KUKA KRL program: EPS_2_25716_MHCR05_A_20250828081216.src

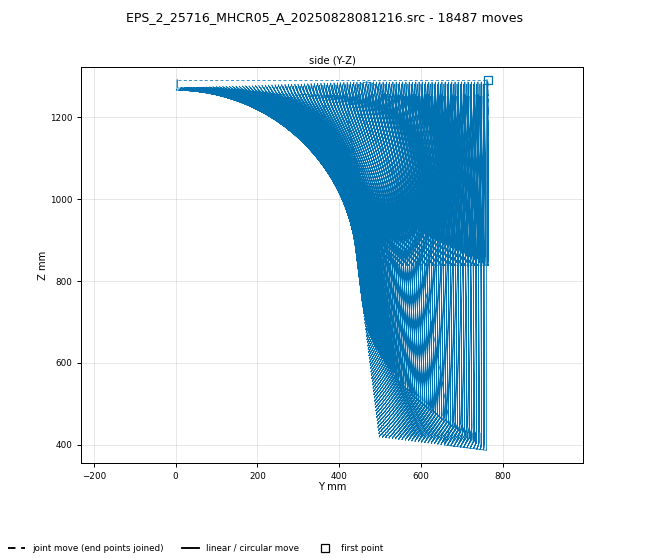
[picture p0: tool path of EPS_2_25716_MHCR05_A_20250828081216.src, 18487 of 18489 moves have a stored position in this frame; points joined in program order, loops and branches not executed]
&ACCESS RVP
&REL 4
&COMMENT QRS 19112012
&PARAM EDITMASK = *
DEF PART()
EXT BAS (BAS_COMMAND :IN,REAL :IN )
INT I
BAS (#INITMOV,0 )

;KUKA QRS Post kuka4.cps  Date:22-06-2017 !

File_ID=2804

QRS_PRE_INIT()

;Init var - Until changes are made in qrs_pre_init
Outlet_Square_prg=0
Inlet_1_Square_prg=0
Inlet_2_Square_prg=0
Inlet_3_Square_prg=0
Inlet_4_Square_prg=0
Inlet_5_Square_prg=0

Outlet_1={X 0.000, Y 457.000, Z 863.000, B 0.000, E1 0.000 }
Inlet_1={X 0.000, Y 457.000, Z 833.000, B 0.000, E1 180.000 }
Outlet_1_type=838
Inlet_1_type=838
;QRS#1=Sidecore dimensions
;QRS#2=825-33" Concrete
;QRS#3=825-33" Concrete
;QRS#4=
;QRS#5=
;QRS#6=
;QRS#7=
;QRS#8=
;QRS#9=S306-46
;QRS#10=S306-46
;QRS#11=
;QRS#12=
;QRS#13=
;QRS#14=
;QRS#15=
;QRS#16=1524x152x1753 5,75'
;QRS#17=EPS Height
;QRS#18=1282
;QRS#19=*
;QRS#20= UPDATED VERSION 22-06-2017
;QRS#21=*
Outlet_Square=0650
Inlet_1_Square=0650
Inlet_2_Square=0
Inlet_3_Square=0
Inlet_4_Square=0
Inlet_5_Square=0
Mill_Square=1
Outlet_Square_Prg=267
Inlet_1_Square_prg=267

QRS_INIT()

$ADVANCE=5

; T1
PTP {E1 177.513,E2 177.513}
PTP {X 0,Y 762.785,A -85,B 0,C 180,E1 177.513,E2 177.513,E3 0,E4 0,E5 0,E6 0}
QRS_SPEED_INIT()
LIN {X 0,Y 762.785,Z 1292,A -85,B 0,C 180,E1 177.513,E2 177.513,E3 0,E4 0,E5 0,E6 0} C_VEL
LIN {X 0,Y 762.785,Z 841.06,A -85,B 0,C 180,E1 177.513,E2 177.513} C_VEL
LIN {X 0,Y 762.866,Z 839.06,A -85,B 0,C 180,E1 177.663,E2 177.663} C_VEL
LIN {X 0,Y 763.878,Z 839.06,A -85,B 0,C 180,E1 179.063,E2 179.063} C_VEL
LIN {X 0,Y 763.781,Z 839.06,A -85,B 0,C 180,E1 186.577,E2 186.577} C_VEL
LIN {X 0,Y 763.753,Z 839.06,A -85,B 0,C 180,E1 194.208,E2 194.208} C_VEL
LIN {X 0,Y 763.775,Z 839.06,A -85,B 0,C 180,E1 202.107,E2 202.107} C_VEL
LIN {X 0,Y 762.947,Z 839.06,A -85,B 0,C 180,E1 208.361,E2 208.361} C_VEL
LIN {X 0,Y 763.678,Z 839.06,A -85,B 0,C 180,E1 209.865,E2 209.865} C_VEL
LIN {X 0,Y 763.751,Z 839.06,A -85,B 0,C 180,E1 217.259,E2 217.259} C_VEL
LIN {X 0,Y 762.19,Z 839.06,A -85,B 0,C 180,E1 222.241,E2 222.241} C_VEL
LIN {X 0,Y 763.489,Z 839.06,A -85,B 0,C 180,E1 224.736,E2 224.736} C_VEL
LIN {X 0,Y 763.718,Z 839.06,A -85,B 0,C 180,E1 225.289,E2 225.289} C_VEL
LIN {X 0,Y 763.691,Z 839.06,A -85,B 0,C 180,E1 233.306,E2 233.306} C_VEL
LIN {X 0,Y 763.599,Z 839.06,A -85,B 0,C 180,E1 233.585,E2 233.585} C_VEL
LIN {X 0,Y 763.105,Z 842.178,A -85,B 0,C 180,E1 233.692,E2 233.692} C_VEL
LIN {X 0,Y 763.151,Z 902.432,A -85,B 0,C 180,E1 234.391,E2 234.391} C_VEL
LIN {X 0,Y 763.569,Z 919.488,A -85,B 0,C 180,E1 234.674,E2 234.674} C_VEL
LIN {X 0,Y 763.689,Z 936.684,A -85,B 0,C 180,E1 235.004,E2 235.004} C_VEL
LIN {X 0,Y 763.627,Z 953.994,A -85,B 0,C 180,E1 235.388,E2 235.388} C_VEL
LIN {X 0,Y 763.298,Z 971.622,A -85,B 0,C 180,E1 235.836,E2 235.836} C_VEL
LIN {X 0,Y 763.66,Z 994.06,A -85,B 0,C 180,E1 236.546,E2 236.546} C_VEL
LIN {X 0,Y 763.665,Z 1012.884,A -85,B 0,C 180,E1 237.214,E2 237.214} C_VEL
LIN {X 0,Y 763.649,Z 1032.465,A -85,B 0,C 180,E1 238,E2 238} C_VEL
LIN {X 0,Y 763.47,Z 1045.091,A -85,B 0,C 180,E1 238.553,E2 238.553} C_VEL
LIN {X 0,Y 763.557,Z 1053.715,A -85,B 0,C 180,E1 238.962,E2 238.962} C_VEL
LIN {X 0,Y 763.507,Z 1068.148,A -85,B 0,C 180,E1 239.675,E2 239.675} C_VEL
LIN {X 0,Y 763.465,Z 1085.374,A -85,B 0,C 180,E1 240.61,E2 240.61} C_VEL
LIN {X 0,Y 763.616,Z 1101.645,A -85,B 0,C 180,E1 241.581,E2 241.581} C_VEL
LIN {X 0,Y 763.575,Z 1117.447,A -85,B 0,C 180,E1 242.599,E2 242.599} C_VEL
LIN {X 0,Y 763.286,Z 1132.483,A -85,B 0,C 180,E1 243.639,E2 243.639} C_VEL
LIN {X 0,Y 763.185,Z 1147.05,A -85,B 0,C 180,E1 244.739,E2 244.739} C_VEL
LIN {X 0,Y 763.452,Z 1160.517,A -85,B 0,C 180,E1 245.849,E2 245.849} C_VEL
LIN {X 0,Y 763.696,Z 1173.568,A -85,B 0,C 180,E1 247.008,E2 247.008} C_VEL
LIN {X 0,Y 763.172,Z 1187.049,A -85,B 0,C 180,E1 248.284,E2 248.284} C_VEL
LIN {X 0,Y 762.923,Z 1198.82,A -85,B 0,C 180,E1 249.499,E2 249.499} C_VEL
LIN {X 0,Y 763.252,Z 1210.585,A -85,B 0,C 180,E1 250.839,E2 250.839} C_VEL
LIN {X 0,Y 763.819,Z 1221.039,A -85,B 0,C 180,E1 252.14,E2 252.14} C_VEL
LIN {X 0,Y 763.048,Z 1231.864,A -85,B 0,C 180,E1 253.594,E2 253.594} C_VEL
LIN {X 0,Y 762.736,Z 1241.602,A -85,B 0,C 180,E1 255.059,E2 255.059} C_VEL
LIN {X 0,Y 763.109,Z 1249.379,A -85,B 0,C 180,E1 256.364,E2 256.364} C_VEL
LIN {X 0,Y 763.845,Z 1256.57,A -85,B 0,C 180,E1 257.724,E2 257.724} C_VEL
LIN {X 0,Y 762.883,Z 1264.428,A -85,B 0,C 180,E1 259.384,E2 259.384} C_VEL
LIN {X 0,Y 762.623,Z 1269.209,A -85,B 0,C 180,E1 260.572,E2 260.572} C_VEL
LIN {X 0,Y 762.835,Z 1272.583,A -85,B 0,C 180,E1 261.525,E2 261.525} C_VEL
LIN {X 0,Y 763.28,Z 1275.723,A -85,B 0,C 180,E1 262.478,E2 262.478} C_VEL
LIN {X 0,Y 763.858,Z 1278.353,A -85,B 0,C 180,E1 263.428,E2 263.428} C_VEL
LIN {X 0,Y 763.258,Z 1280.666,A -85,B 0,C 180,E1 264.366,E2 264.366} C_VEL
LIN {X 0,Y 762.774,Z 1282.62,A -85,B 0,C 180,E1 265.305,E2 265.305} C_VEL
LIN {X 0,Y 762.587,Z 1284.207,A -85,B 0,C 180,E1 266.245,E2 266.245} C_VEL
LIN {X 0,Y 762.778,Z 1285.378,A -85,B 0,C 180,E1 267.186,E2 267.186} C_VEL
LIN {X 0,Y 763.829,Z 1286.67,A -85,B 0,C 180,E1 269.066,E2 269.066} C_VEL
LIN {X 0,Y 762.793,Z 1286.715,A -85,B 0,C 180,E1 270.942,E2 270.942} C_VEL
LIN {X 0,Y 762.612,Z 1286.489,A -85,B 0,C 180,E1 271.58,E2 271.58} C_VEL
LIN {X 0,Y 762.793,Z 1285.372,A -85,B 0,C 180,E1 272.82,E2 272.82} C_VEL
LIN {X 0,Y 763.264,Z 1284.181,A -85,B 0,C 180,E1 273.758,E2 273.758} C_VEL
LIN {X 0,Y 763.868,Z 1282.57,A -85,B 0,C 180,E1 274.695,E2 274.695} C_VEL
LIN {X 0,Y 763.015,Z 1279.579,A -85,B 0,C 180,E1 276.114,E2 276.114} C_VEL
LIN {X 0,Y 762.631,Z 1275.706,A -85,B 0,C 180,E1 277.536,E2 277.536} C_VEL
LIN {X 0,Y 763.011,Z 1270.959,A -85,B 0,C 180,E1 278.954,E2 278.954} C_VEL
LIN {X 0,Y 763.87,Z 1265.354,A -85,B 0,C 180,E1 280.37,E2 280.37} C_VEL
LIN {X 0,Y 763.474,Z 1262.202,A -85,B 0,C 180,E1 281.092,E2 281.092} C_VEL
LIN {X 0,Y 762.849,Z 1256.532,A -85,B 0,C 180,E1 282.299,E2 282.299} C_VEL
LIN {X 0,Y 762.722,Z 1249.063,A -85,B 0,C 180,E1 283.698,E2 283.698} C_VEL
LIN {X 0,Y 763.275,Z 1240.923,A -85,B 0,C 180,E1 285.043,E2 285.043} C_VEL
LIN {X 0,Y 763.758,Z 1235.327,A -85,B 0,C 180,E1 285.873,E2 285.873} C_VEL
LIN {X 0,Y 763.633,Z 1231.816,A -85,B 0,C 180,E1 286.4,E2 286.4} C_VEL
LIN {X 0,Y 762.911,Z 1220.984,A -85,B 0,C 180,E1 287.889,E2 287.889} C_VEL
LIN {X 0,Y 762.868,Z 1209,A -85,B 0,C 180,E1 289.358,E2 289.358} C_VEL
LIN {X 0,Y 763.421,Z 1197.407,A -85,B 0,C 180,E1 290.64,E2 290.64} C_VEL
LIN {X 0,Y 763.771,Z 1189.172,A -85,B 0,C 180,E1 291.478,E2 291.478} C_VEL
LIN {X 0,Y 763.561,Z 1182.825,A -85,B 0,C 180,E1 292.116,E2 292.116} C_VEL
LIN {X 0,Y 763.219,Z 1172.077,A -85,B 0,C 180,E1 293.142,E2 293.142} C_VEL
LIN {X 0,Y 763.156,Z 1158.949,A -85,B 0,C 180,E1 294.293,E2 294.293} C_VEL
LIN {X 0,Y 763.463,Z 1145.228,A -85,B 0,C 180,E1 295.394,E2 295.394} C_VEL
LIN {X 0,Y 763.662,Z 1130.565,A -85,B 0,C 180,E1 296.486,E2 296.486} C_VEL
LIN {X 0,Y 763.467,Z 1114.323,A -85,B 0,C 180,E1 297.612,E2 297.612} C_VEL
LIN {X 0,Y 763.401,Z 1098.789,A -85,B 0,C 180,E1 298.602,E2 298.602} C_VEL
LIN {X 0,Y 763.564,Z 1082.344,A -85,B 0,C 180,E1 299.557,E2 299.557} C_VEL
LIN {X 0,Y 763.601,Z 1066.411,A -85,B 0,C 180,E1 300.413,E2 300.413} C_VEL
LIN {X 0,Y 763.622,Z 1047.439,A -85,B 0,C 180,E1 301.337,E2 301.337} C_VEL
LIN {X 0,Y 763.594,Z 1028.686,A -85,B 0,C 180,E1 302.161,E2 302.161} C_VEL
LIN {X 0,Y 763.579,Z 1010.173,A -85,B 0,C 180,E1 302.89,E2 302.89} C_VEL
LIN {X 0,Y 763.358,Z 997.463,A -85,B 0,C 180,E1 303.349,E2 303.349} C_VEL
LIN {X 0,Y 763.576,Z 988.896,A -85,B 0,C 180,E1 303.623,E2 303.623} C_VEL
LIN {X 0,Y 763.726,Z 970.079,A -85,B 0,C 180,E1 304.185,E2 304.185} C_VEL
LIN {X 0,Y 763.711,Z 953.48,A -85,B 0,C 180,E1 304.621,E2 304.621} C_VEL
LIN {X 0,Y 763.519,Z 936.23,A -85,B 0,C 180,E1 305.015,E2 305.015} C_VEL
LIN {X 0,Y 763.194,Z 924.975,A -85,B 0,C 180,E1 305.251,E2 305.251} C_VEL
LIN {X 0,Y 763.49,Z 908.084,A -85,B 0,C 180,E1 305.51,E2 305.51} C_VEL
LIN {X 0,Y 763.502,Z 896.075,A -85,B 0,C 180,E1 305.669,E2 305.669} C_VEL
LIN {X 0,Y 763.101,Z 839.511,A -85,B 0,C 180,E1 306.339,E2 306.339} C_VEL
LIN {X 0,Y 763.718,Z 839.06,A -85,B 0,C 180,E1 306.442,E2 306.442} C_VEL
LIN {X 0,Y 763.692,Z 839.06,A -85,B 0,C 180,E1 306.694,E2 306.694} C_VEL
LIN {X 0,Y 763.713,Z 839.06,A -85,B 0,C 180,E1 314.721,E2 314.721} C_VEL
LIN {X 0,Y 763.497,Z 839.06,A -85,B 0,C 180,E1 315.265,E2 315.265} C_VEL
LIN {X 0,Y 762.413,Z 839.06,A -85,B 0,C 180,E1 320.391,E2 320.391} C_VEL
LIN {X 0,Y 763.779,Z 839.06,A -85,B 0,C 180,E1 322.742,E2 322.742} C_VEL
LIN {X 0,Y 763.789,Z 839.06,A -85,B 0,C 180,E1 329.521,E2 329.521} C_VEL
LIN {X 0,Y 763.786,Z 839.06,A -85,B 0,C 180,E1 335.855,E2 335.855} C_VEL
LIN {X 0,Y 763.81,Z 839.06,A -85,B 0,C 180,E1 343.85,E2 343.85} C_VEL
LIN {X 0,Y 763.85,Z 839.06,A -85,B 0,C 180,E1 351.533,E2 351.533} C_VEL
LIN {X 0,Y 763.887,Z 839.06,A -85,B 0,C 180,E1 359.063,E2 359.063} C_VEL
LIN {X 0,Y 763.839,Z 839.06,A -85,B 0,C 180,E1 366.576,E2 366.576} C_VEL
LIN {X 0,Y 763.861,Z 839.06,A -85,B 0,C 180,E1 374.206,E2 374.206} C_VEL
LIN {X 0,Y 763.821,Z 839.06,A -85,B 0,C 180,E1 382.105,E2 382.105} C_VEL
LIN {X 0,Y 762.949,Z 839.06,A -85,B 0,C 180,E1 388.361,E2 388.361} C_VEL
LIN {X 0,Y 763.665,Z 839.06,A -85,B 0,C 180,E1 389.85,E2 389.85} C_VEL
LIN {X 0,Y 763.783,Z 839.06,A -85,B 0,C 180,E1 397.257,E2 397.257} C_VEL
LIN {X 0,Y 762.287,Z 839.06,A -85,B 0,C 180,E1 402.459,E2 402.459} C_VEL
LIN {X 0,Y 763.519,Z 839.06,A -85,B 0,C 180,E1 404.734,E2 404.734} C_VEL
LIN {X 0,Y 763.736,Z 839.06,A -85,B 0,C 180,E1 405.281,E2 405.281} C_VEL
LIN {X 0,Y 763.707,Z 839.06,A -85,B 0,C 180,E1 413.304,E2 413.304} C_VEL
LIN {X 0,Y 763.661,Z 839.06,A -85,B 0,C 180,E1 413.601,E2 413.601} C_VEL
LIN {X 0,Y 761.689,Z 839.06,A -85,B 0,C 180,E1 413.812,E2 413.812} C_VEL
LIN {X 0,Y 761.812,Z 840.818,A -85,B 0,C 180,E1 413.903,E2 413.903} C_VEL
LIN {X 0,Y 762.77,Z 843.615,A -85,B 0,C 180,E1 413.987,E2 413.987} C_VEL
LIN {X 0,Y 763.13,Z 845.592,A -85,B 0,C 180,E1 414.029,E2 414.029} C_VEL
LIN {X 0,Y 763.65,Z 875.73,A -85,B 0,C 180,E1 414.419,E2 414.419} C_VEL
LIN {X 0,Y 763.658,Z 892.175,A -85,B 0,C 180,E1 414.679,E2 414.679} C_VEL
LIN {X 0,Y 763.408,Z 909.107,A -85,B 0,C 180,E1 414.995,E2 414.995} C_VEL
LIN {X 0,Y 763.241,Z 916.55,A -85,B 0,C 180,E1 415.149,E2 415.149} C_VEL
LIN {X 0,Y 763.606,Z 932.664,A -85,B 0,C 180,E1 415.562,E2 415.562} C_VEL
LIN {X 0,Y 763.666,Z 945.84,A -85,B 0,C 180,E1 415.934,E2 415.934} C_VEL
LIN {X 0,Y 763.644,Z 964.876,A -85,B 0,C 180,E1 416.529,E2 416.529} C_VEL
LIN {X 0,Y 763.371,Z 982.796,A -85,B 0,C 180,E1 417.152,E2 417.152} C_VEL
LIN {X 0,Y 763.602,Z 1002.249,A -85,B 0,C 180,E1 417.944,E2 417.944} C_VEL
LIN {X 0,Y 763.603,Z 1020.397,A -85,B 0,C 180,E1 418.756,E2 418.756} C_VEL
LIN {X 0,Y 763.645,Z 1038.535,A -85,B 0,C 180,E1 419.657,E2 419.657} C_VEL
LIN {X 0,Y 763.579,Z 1054.594,A -85,B 0,C 180,E1 420.524,E2 420.524} C_VEL
LIN {X 0,Y 763.423,Z 1071.141,A -85,B 0,C 180,E1 421.496,E2 421.496} C_VEL
LIN {X 0,Y 763.34,Z 1087.981,A -85,B 0,C 180,E1 422.582,E2 422.582} C_VEL
LIN {X 0,Y 763.549,Z 1102.977,A -85,B 0,C 180,E1 423.641,E2 423.641} C_VEL
LIN {X 0,Y 763.649,Z 1117.051,A -85,B 0,C 180,E1 424.71,E2 424.71} C_VEL
LIN {X 0,Y 763.257,Z 1130.941,A -85,B 0,C 180,E1 425.835,E2 425.835} C_VEL
LIN {X 0,Y 763.008,Z 1143.961,A -85,B 0,C 180,E1 426.978,E2 426.978} C_VEL
LIN {X 0,Y 763.296,Z 1157.072,A -85,B 0,C 180,E1 428.245,E2 428.245} C_VEL
LIN {X 0,Y 763.8,Z 1169.152,A -85,B 0,C 180,E1 429.516,E2 429.516} C_VEL
LIN {X 0,Y 763.197,Z 1180.742,A -85,B 0,C 180,E1 430.812,E2 430.812} C_VEL
LIN {X 0,Y 762.792,Z 1191.318,A -85,B 0,C 180,E1 432.108,E2 432.108} C_VEL
LIN {X 0,Y 763.104,Z 1202.116,A -85,B 0,C 180,E1 433.588,E2 433.588} C_VEL
LIN {X 0,Y 763.757,Z 1210.687,A -85,B 0,C 180,E1 434.883,E2 434.883} C_VEL
LIN {X 0,Y 763.675,Z 1213.295,A -85,B 0,C 180,E1 435.315,E2 435.315} C_VEL
LIN {X 0,Y 763.015,Z 1219.935,A -85,B 0,C 180,E1 436.42,E2 436.42} C_VEL
LIN {X 0,Y 762.583,Z 1227.944,A -85,B 0,C 180,E1 437.937,E2 437.937} C_VEL
LIN {X 0,Y 762.996,Z 1234.58,A -85,B 0,C 180,E1 439.379,E2 439.379} C_VEL
LIN {X 0,Y 763.697,Z 1239.36,A -85,B 0,C 180,E1 440.579,E2 440.579} C_VEL
LIN {X 0,Y 763.674,Z 1241.105,A -85,B 0,C 180,E1 441.053,E2 441.053} C_VEL
LIN {X 0,Y 762.88,Z 1245.837,A -85,B 0,C 180,E1 442.467,E2 442.467} C_VEL
LIN {X 0,Y 762.627,Z 1249.69,A -85,B 0,C 180,E1 443.882,E2 443.882} C_VEL
LIN {X 0,Y 763.151,Z 1252.687,A -85,B 0,C 180,E1 445.3,E2 445.3} C_VEL
LIN {X 0,Y 763.839,Z 1254.408,A -85,B 0,C 180,E1 446.388,E2 446.388} C_VEL
LIN {X 0,Y 763.401,Z 1255.391,A -85,B 0,C 180,E1 447.182,E2 447.182} C_VEL
LIN {X 0,Y 762.542,Z 1256.734,A -85,B 0,C 180,E1 449.058,E2 449.058} C_VEL
LIN {X 0,Y 762.958,Z 1256.698,A -85,B 0,C 180,E1 450.935,E2 450.935} C_VEL
LIN {X 0,Y 763.557,Z 1255.31,A -85,B 0,C 180,E1 452.811,E2 452.811} C_VEL
LIN {X 0,Y 762.975,Z 1254.137,A -85,B 0,C 180,E1 453.753,E2 453.753} C_VEL
LIN {X 0,Y 762.645,Z 1252.533,A -85,B 0,C 180,E1 454.696,E2 454.696} C_VEL
LIN {X 0,Y 762.762,Z 1249.484,A -85,B 0,C 180,E1 456.11,E2 456.11} C_VEL
LIN {X 0,Y 763.538,Z 1245.587,A -85,B 0,C 180,E1 457.52,E2 457.52} C_VEL
LIN {X 0,Y 763.844,Z 1244.019,A -85,B 0,C 180,E1 457.99,E2 457.99} C_VEL
LIN {X 0,Y 763.275,Z 1240.83,A -85,B 0,C 180,E1 458.944,E2 458.944} C_VEL
LIN {X 0,Y 762.602,Z 1234.243,A -85,B 0,C 180,E1 460.62,E2 460.62} C_VEL
LIN {X 0,Y 762.993,Z 1226.33,A -85,B 0,C 180,E1 462.29,E2 462.29} C_VEL
LIN {X 0,Y 763.73,Z 1219.455,A -85,B 0,C 180,E1 463.566,E2 463.566} C_VEL
LIN {X 0,Y 763.759,Z 1217.556,A -85,B 0,C 180,E1 463.884,E2 463.884} C_VEL
LIN {X 0,Y 763.136,Z 1210.866,A -85,B 0,C 180,E1 465.01,E2 465.01} C_VEL
LIN {X 0,Y 762.705,Z 1201.563,A -85,B 0,C 180,E1 466.414,E2 466.414} C_VEL
LIN {X 0,Y 763.094,Z 1189.694,A -85,B 0,C 180,E1 468.001,E2 468.001} C_VEL
LIN {X 0,Y 763.767,Z 1179.038,A -85,B 0,C 180,E1 469.285,E2 469.285} C_VEL
LIN {X 0,Y 763.28,Z 1167.08,A -85,B 0,C 180,E1 470.632,E2 470.632} C_VEL
LIN {X 0,Y 762.97,Z 1155.209,A -85,B 0,C 180,E1 471.862,E2 471.862} C_VEL
LIN {X 0,Y 763.232,Z 1141.649,A -85,B 0,C 180,E1 473.135,E2 473.135} C_VEL
LIN {X 0,Y 763.679,Z 1128.165,A -85,B 0,C 180,E1 474.294,E2 474.294} C_VEL
LIN {X 0,Y 763.562,Z 1116.121,A -85,B 0,C 180,E1 475.278,E2 475.278} C_VEL
LIN {X 0,Y 763.276,Z 1100.026,A -85,B 0,C 180,E1 476.492,E2 476.492} C_VEL
LIN {X 0,Y 763.361,Z 1084.775,A -85,B 0,C 180,E1 477.542,E2 477.542} C_VEL
LIN {X 0,Y 763.577,Z 1068.971,A -85,B 0,C 180,E1 478.539,E2 478.539} C_VEL
LIN {X 0,Y 763.632,Z 1051.912,A -85,B 0,C 180,E1 479.532,E2 479.532} C_VEL
LIN {X 0,Y 763.542,Z 1035.674,A -85,B 0,C 180,E1 480.407,E2 480.407} C_VEL
LIN {X 0,Y 763.571,Z 1017.254,A -85,B 0,C 180,E1 481.302,E2 481.302} C_VEL
LIN {X 0,Y 763.523,Z 998.236,A -85,B 0,C 180,E1 482.137,E2 482.137} C_VEL
LIN {X 0,Y 763.43,Z 991.336,A -85,B 0,C 180,E1 482.416,E2 482.416} C_VEL
LIN {X 0,Y 763.663,Z 979.229,A -85,B 0,C 180,E1 482.874,E2 482.874} C_VEL
LIN {X 0,Y 763.696,Z 961.114,A -85,B 0,C 180,E1 483.504,E2 483.504} C_VEL
LIN {X 0,Y 763.649,Z 940.7,A -85,B 0,C 180,E1 484.127,E2 484.127} C_VEL
LIN {X 0,Y 763.287,Z 923.063,A -85,B 0,C 180,E1 484.608,E2 484.608} C_VEL
LIN {X 0,Y 763.424,Z 916.043,A -85,B 0,C 180,E1 484.763,E2 484.763} C_VEL
LIN {X 0,Y 763.72,Z 898.672,A -85,B 0,C 180,E1 485.108,E2 485.108} C_VEL
LIN {X 0,Y 763.762,Z 883.162,A -85,B 0,C 180,E1 485.376,E2 485.376} C_VEL
LIN {X 0,Y 763.655,Z 867.28,A -85,B 0,C 180,E1 485.601,E2 485.601} C_VEL
LIN {X 0,Y 763.073,Z 839.454,A -85,B 0,C 180,E1 485.954,E2 485.954} C_VEL
LIN {X 0,Y 763.407,Z 839.06,A -85,B 0,C 180,E1 486,E2 486} C_VEL
LIN {X 0,Y 763.84,Z 839.06,A -85,B 0,C 180,E1 486.105,E2 486.105} C_VEL
LIN {X 0,Y 763.699,Z 839.06,A -85,B 0,C 180,E1 486.718,E2 486.718} C_VEL
LIN {X 0,Y 763.708,Z 839.06,A -85,B 0,C 180,E1 494.712,E2 494.712} C_VEL
LIN {X 0,Y 763.492,Z 839.06,A -85,B 0,C 180,E1 495.264,E2 495.264} C_VEL
LIN {X 0,Y 762.398,Z 839.06,A -85,B 0,C 180,E1 500.382,E2 500.382} C_VEL
LIN {X 0,Y 763.769,Z 839.06,A -85,B 0,C 180,E1 502.742,E2 502.742} C_VEL
LIN {X 0,Y 763.674,Z 839.06,A -85,B 0,C 180,E1 510.135,E2 510.135} C_VEL
LIN {X 0,Y 762.95,Z 839.06,A -85,B 0,C 180,E1 511.639,E2 511.639} C_VEL
LIN {X 0,Y 763.788,Z 839.06,A -85,B 0,C 180,E1 517.894,E2 517.894} C_VEL
LIN {X 0,Y 763.46,Z 839.06,A -85,B 0,C 180,E1 524.94,E2 524.94} C_VEL
LIN {X 0,Y 763.555,Z 839.06,A -85,B 0,C 180,E1 525.788,E2 525.788} C_VEL
LIN {X 0,Y 763.79,Z 839.06,A -85,B 0,C 180,E1 531.532,E2 531.532} C_VEL
LIN {X 0,Y 762.866,Z 839.06,A -85,B 0,C 180,E1 537.663,E2 537.663} C_VEL
LIN {X 0,Y 754.969,Z 839.06,A -85,B 0,C 180,E1 540.292,E2 540.292} C_VEL
LIN {X 0,Y 755.025,Z 839.06,A -85,B 0,C 180,E1 547.538,E2 547.538} C_VEL
LIN {X 0,Y 754.615,Z 839.06,A -85,B 0,C 180,E1 555.783,E2 555.783} C_VEL
LIN {X 0,Y 755.029,Z 839.06,A -85,B 0,C 180,E1 563.105,E2 563.105} C_VEL
LIN {X 0,Y 754.735,Z 839.06,A -85,B 0,C 180,E1 571.255,E2 571.255} C_VEL
LIN {X 0,Y 755.273,Z 839.06,A -85,B 0,C 180,E1 577.826,E2 577.826} C_VEL
LIN {X 0,Y 755.063,Z 839.06,A -85,B 0,C 180,E1 586.081,E2 586.081} C_VEL
LIN {X 0,Y 755.753,Z 840.318,A -85,B 0,C 180,E1 593.259,E2 593.259} C_VEL
LIN {X 0,Y 757.074,Z 944.077,A -85,B 0,C 180,E1 594.812,E2 594.812} C_VEL
LIN {X 0,Y 756.745,Z 1014.661,A -85,B 0,C 180,E1 596.948,E2 596.948} C_VEL
LIN {X 0,Y 756.205,Z 1085.22,A -85,B 0,C 180,E1 600.29,E2 600.29} C_VEL
LIN {X 0,Y 755.603,Z 1150.188,A -85,B 0,C 180,E1 604.727,E2 604.727} C_VEL
LIN {X 0,Y 755.136,Z 1202.606,A -85,B 0,C 180,E1 609.709,E2 609.709} C_VEL
LIN {X 0,Y 754.862,Z 1239.376,A -85,B 0,C 180,E1 614.546,E2 614.546} C_VEL
LIN {X 0,Y 754.828,Z 1265.626,A -85,B 0,C 180,E1 619.572,E2 619.572} C_VEL
LIN {X 0,Y 755.018,Z 1281.752,A -85,B 0,C 180,E1 624.809,E2 624.809} C_VEL
LIN {X 0,Y 754.933,Z 1286.837,A -85,B 0,C 180,E1 630.576,E2 630.576} C_VEL
LIN {X 0,Y 755.217,Z 1280.596,A -85,B 0,C 180,E1 635.73,E2 635.73} C_VEL
LIN {X 0,Y 755.2,Z 1260.438,A -85,B 0,C 180,E1 641.597,E2 641.597} C_VEL
LIN {X 0,Y 755.263,Z 1226.677,A -85,B 0,C 180,E1 647.299,E2 647.299} C_VEL
LIN {X 0,Y 755.617,Z 1178.746,A -85,B 0,C 180,E1 652.753,E2 652.753} C_VEL
LIN {X 0,Y 756.04,Z 1119.014,A -85,B 0,C 180,E1 657.587,E2 657.587} C_VEL
LIN {X 0,Y 756.523,Z 1050.346,A -85,B 0,C 180,E1 661.527,E2 661.527} C_VEL
LIN {X 0,Y 756.942,Z 978.376,A -85,B 0,C 180,E1 664.286,E2 664.286} C_VEL
LIN {X 0,Y 756.999,Z 905.014,A -85,B 0,C 180,E1 665.907,E2 665.907} C_VEL
LIN {X 0,Y 755.594,Z 839.06,A -85,B 0,C 180,E1 666.793,E2 666.793} C_VEL
LIN {X 0,Y 754.921,Z 839.06,A -85,B 0,C 180,E1 676.058,E2 676.058} C_VEL
LIN {X 0,Y 755.19,Z 839.06,A -85,B 0,C 180,E1 683.613,E2 683.613} C_VEL
LIN {X 0,Y 754.947,Z 839.06,A -85,B 0,C 180,E1 691.015,E2 691.015} C_VEL
LIN {X 0,Y 754.939,Z 839.06,A -85,B 0,C 180,E1 696.892,E2 696.892} C_VEL
LIN {X 0,Y 755.476,Z 839.06,A -85,B 0,C 180,E1 704.235,E2 704.235} C_VEL
LIN {X 0,Y 755.156,Z 839.06,A -85,B 0,C 180,E1 712.463,E2 712.463} C_VEL
LIN {X 0,Y 754.846,Z 839.06,A -85,B 0,C 180,E1 720.543,E2 720.543} C_VEL
LIN {X 0,Y 755.135,Z 839.06,A -85,B 0,C 180,E1 727.471,E2 727.471} C_VEL
LIN {X 0,Y 754.737,Z 839.06,A -85,B 0,C 180,E1 735.712,E2 735.712} C_VEL
LIN {X 0,Y 755.112,Z 839.06,A -85,B 0,C 180,E1 743.031,E2 743.031} C_VEL
LIN {X 0,Y 754.707,Z 839.06,A -85,B 0,C 180,E1 751.251,E2 751.251} C_VEL
LIN {X 0,Y 755.383,Z 839.06,A -85,B 0,C 180,E1 757.735,E2 757.735} C_VEL
LIN {X 0,Y 755.05,Z 839.06,A -85,B 0,C 180,E1 766.079,E2 766.079} C_VEL
LIN {X 0,Y 755.012,Z 839.06,A -85,B 0,C 180,E1 773.483,E2 773.483} C_VEL
LIN {X 0,Y 756.859,Z 930.469,A -85,B 0,C 180,E1 775.155,E2 775.155} C_VEL
LIN {X 0,Y 756.556,Z 1006.275,A -85,B 0,C 180,E1 777.791,E2 777.791} C_VEL
LIN {X 0,Y 756.005,Z 1077.386,A -85,B 0,C 180,E1 781.597,E2 781.597} C_VEL
LIN {X 0,Y 755.422,Z 1139.164,A -85,B 0,C 180,E1 786.301,E2 786.301} C_VEL
LIN {X 0,Y 755.134,Z 1185.86,A -85,B 0,C 180,E1 791.236,E2 791.236} C_VEL
LIN {X 0,Y 755.113,Z 1220.136,A -85,B 0,C 180,E1 796.314,E2 796.314} C_VEL
LIN {X 0,Y 755.167,Z 1244.31,A -85,B 0,C 180,E1 801.91,E2 801.91} C_VEL
LIN {X 0,Y 755.427,Z 1255.392,A -85,B 0,C 180,E1 807.12,E2 807.12} C_VEL
LIN {X 0,Y 755.499,Z 1255.313,A -85,B 0,C 180,E1 812.879,E2 812.879} C_VEL
LIN {X 0,Y 755.449,Z 1242.067,A -85,B 0,C 180,E1 818.668,E2 818.668} C_VEL
LIN {X 0,Y 755.414,Z 1214.542,A -85,B 0,C 180,E1 824.549,E2 824.549} C_VEL
LIN {X 0,Y 755.564,Z 1172.21,A -85,B 0,C 180,E1 830.279,E2 830.279} C_VEL
LIN {X 0,Y 755.958,Z 1117.716,A -85,B 0,C 180,E1 835.42,E2 835.42} C_VEL
LIN {X 0,Y 756.368,Z 1053.011,A -85,B 0,C 180,E1 839.786,E2 839.786} C_VEL
LIN {X 0,Y 756.769,Z 981.361,A -85,B 0,C 180,E1 843.137,E2 843.137} C_VEL
LIN {X 0,Y 757.059,Z 905.851,A -85,B 0,C 180,E1 845.321,E2 845.321} C_VEL
LIN {X 0,Y 755.773,Z 839.06,A -85,B 0,C 180,E1 846.428,E2 846.428} C_VEL
LIN {X 0,Y 755.303,Z 839.06,A -85,B 0,C 180,E1 855.522,E2 855.522} C_VEL
LIN {X 0,Y 755.064,Z 839.06,A -85,B 0,C 180,E1 863.688,E2 863.688} C_VEL
LIN {X 0,Y 754.83,Z 839.06,A -85,B 0,C 180,E1 871.851,E2 871.851} C_VEL
LIN {X 0,Y 754.723,Z 839.06,A -85,B 0,C 180,E1 879.438,E2 879.438} C_VEL
LIN {X 0,Y 754.887,Z 839.06,A -85,B 0,C 180,E1 887.253,E2 887.253} C_VEL
LIN {X 0,Y 755.036,Z 839.06,A -85,B 0,C 180,E1 892.528,E2 892.528} C_VEL
LIN {X 0,Y 754.969,Z 839.06,A -85,B 0,C 180,E1 900.292,E2 900.292} C_VEL
LIN {X 0,Y 746.202,Z 839.06,A -85,B 0,C 180,E1 902.918,E2 902.918} C_VEL
LIN {X 0,Y 746.963,Z 839.06,A -85,B 0,C 180,E1 907.62,E2 907.62} C_VEL
LIN {X 0,Y 747.02,Z 839.06,A -85,B 0,C 180,E1 915.137,E2 915.137} C_VEL
LIN {X 0,Y 746.898,Z 839.06,A -85,B 0,C 180,E1 923.371,E2 923.371} C_VEL
LIN {X 0,Y 746.735,Z 839.06,A -85,B 0,C 180,E1 931.244,E2 931.244} C_VEL
LIN {X 0,Y 746.82,Z 839.06,A -85,B 0,C 180,E1 938.5,E2 938.5} C_VEL
LIN {X 0,Y 746.975,Z 839.06,A -85,B 0,C 180,E1 946.189,E2 946.189} C_VEL
LIN {X 0,Y 747.305,Z 840.241,A -85,B 0,C 180,E1 952.773,E2 952.773} C_VEL
LIN {X 0,Y 750.255,Z 852.659,A -85,B 0,C 180,E1 953.09,E2 953.09} C_VEL
LIN {X 0,Y 750.475,Z 943.337,A -85,B 0,C 180,E1 954.439,E2 954.439} C_VEL
LIN {X 0,Y 749.879,Z 1014.162,A -85,B 0,C 180,E1 956.585,E2 956.585} C_VEL
LIN {X 0,Y 748.99,Z 1084.695,A -85,B 0,C 180,E1 959.943,E2 959.943} C_VEL
LIN {X 0,Y 747.987,Z 1149.813,A -85,B 0,C 180,E1 964.42,E2 964.42} C_VEL
LIN {X 0,Y 747.293,Z 1201.259,A -85,B 0,C 180,E1 969.331,E2 969.331} C_VEL
LIN {X 0,Y 746.997,Z 1238.916,A -85,B 0,C 180,E1 974.309,E2 974.309} C_VEL
LIN {X 0,Y 746.892,Z 1265.627,A -85,B 0,C 180,E1 979.46,E2 979.46} C_VEL
LIN {X 0,Y 747.054,Z 1281.752,A -85,B 0,C 180,E1 984.754,E2 984.754} C_VEL
LIN {X 0,Y 746.944,Z 1286.837,A -85,B 0,C 180,E1 990.583,E2 990.583} C_VEL
LIN {X 0,Y 747.182,Z 1280.596,A -85,B 0,C 180,E1 995.792,E2 995.792} C_VEL
LIN {X 0,Y 747.188,Z 1260.439,A -85,B 0,C 180,E1 1001.723,E2 1001.723} C_VEL
LIN {X 0,Y 747.388,Z 1227.975,A -85,B 0,C 180,E1 1007.308,E2 1007.308} C_VEL
LIN {X 0,Y 747.871,Z 1179.974,A -85,B 0,C 180,E1 1012.883,E2 1012.883} C_VEL
LIN {X 0,Y 748.581,Z 1120.467,A -85,B 0,C 180,E1 1017.782,E2 1017.782} C_VEL
LIN {X 0,Y 749.458,Z 1051.504,A -85,B 0,C 180,E1 1021.801,E2 1021.801} C_VEL
LIN {X 0,Y 750.198,Z 979.58,A -85,B 0,C 180,E1 1024.6,E2 1024.6} C_VEL
LIN {X 0,Y 750.493,Z 905.856,A -85,B 0,C 180,E1 1026.254,E2 1026.254} C_VEL
LIN {X 0,Y 748.728,Z 843.606,A -85,B 0,C 180,E1 1027.104,E2 1027.104} C_VEL
LIN {X 0,Y 747.071,Z 839.06,A -85,B 0,C 180,E1 1027.419,E2 1027.419} C_VEL
LIN {X 0,Y 746.853,Z 839.06,A -85,B 0,C 180,E1 1036.188,E2 1036.188} C_VEL
LIN {X 0,Y 747.275,Z 839.06,A -85,B 0,C 180,E1 1043.366,E2 1043.366} C_VEL
LIN {X 0,Y 746.809,Z 839.06,A -85,B 0,C 180,E1 1051.445,E2 1051.445} C_VEL
LIN {X 0,Y 746.477,Z 839.06,A -85,B 0,C 180,E1 1057.72,E2 1057.72} C_VEL
LIN {X 0,Y 746.795,Z 839.06,A -85,B 0,C 180,E1 1065.254,E2 1065.254} C_VEL
LIN {X 0,Y 747.179,Z 839.06,A -85,B 0,C 180,E1 1072.382,E2 1072.382} C_VEL
LIN {X 0,Y 746.859,Z 839.06,A -85,B 0,C 180,E1 1080.549,E2 1080.549} C_VEL
LIN {X 0,Y 747.072,Z 839.06,A -85,B 0,C 180,E1 1087.552,E2 1087.552} C_VEL
LIN {X 0,Y 747.095,Z 839.06,A -85,B 0,C 180,E1 1095.156,E2 1095.156} C_VEL
LIN {X 0,Y 746.95,Z 839.06,A -85,B 0,C 180,E1 1103.297,E2 1103.297} C_VEL
LIN {X 0,Y 746.764,Z 839.06,A -85,B 0,C 180,E1 1111.164,E2 1111.164} C_VEL
LIN {X 0,Y 746.844,Z 839.06,A -85,B 0,C 180,E1 1118.501,E2 1118.501} C_VEL
LIN {X 0,Y 747.031,Z 839.06,A -85,B 0,C 180,E1 1126.088,E2 1126.088} C_VEL
LIN {X 0,Y 747.595,Z 840.26,A -85,B 0,C 180,E1 1133.099,E2 1133.099} C_VEL
LIN {X 0,Y 750.535,Z 864.887,A -85,B 0,C 180,E1 1133.557,E2 1133.557} C_VEL
LIN {X 0,Y 750.234,Z 940.158,A -85,B 0,C 180,E1 1135.07,E2 1135.07} C_VEL
LIN {X 0,Y 749.522,Z 1012.551,A -85,B 0,C 180,E1 1137.738,E2 1137.738} C_VEL
LIN {X 0,Y 748.56,Z 1082.96,A -85,B 0,C 180,E1 1141.655,E2 1141.655} C_VEL
LIN {X 0,Y 747.669,Z 1143.719,A -85,B 0,C 180,E1 1146.455,E2 1146.455} C_VEL
LIN {X 0,Y 747.159,Z 1189.701,A -85,B 0,C 180,E1 1151.511,E2 1151.511} C_VEL
LIN {X 0,Y 746.946,Z 1223.011,A -85,B 0,C 180,E1 1156.714,E2 1156.714} C_VEL
LIN {X 0,Y 747.228,Z 1244.309,A -85,B 0,C 180,E1 1161.824,E2 1161.824} C_VEL
LIN {X 0,Y 747.427,Z 1255.392,A -85,B 0,C 180,E1 1167.089,E2 1167.089} C_VEL
LIN {X 0,Y 747.469,Z 1255.313,A -85,B 0,C 180,E1 1172.91,E2 1172.91} C_VEL
LIN {X 0,Y 747.397,Z 1242.069,A -85,B 0,C 180,E1 1178.762,E2 1178.762} C_VEL
LIN {X 0,Y 747.423,Z 1214.547,A -85,B 0,C 180,E1 1184.708,E2 1184.708} C_VEL
LIN {X 0,Y 747.731,Z 1173.565,A -85,B 0,C 180,E1 1190.346,E2 1190.346} C_VEL
LIN {X 0,Y 748.362,Z 1120.038,A -85,B 0,C 180,E1 1195.503,E2 1195.503} C_VEL
LIN {X 0,Y 749.084,Z 1056.777,A -85,B 0,C 180,E1 1199.882,E2 1199.882} C_VEL
LIN {X 0,Y 749.833,Z 985.204,A -85,B 0,C 180,E1 1203.33,E2 1203.33} C_VEL
LIN {X 0,Y 750.395,Z 910.224,A -85,B 0,C 180,E1 1205.589,E2 1205.589} C_VEL
LIN {X 0,Y 748.585,Z 842.763,A -85,B 0,C 180,E1 1206.725,E2 1206.725} C_VEL
LIN {X 0,Y 747.501,Z 839.06,A -85,B 0,C 180,E1 1206.936,E2 1206.936} C_VEL
LIN {X 0,Y 746.839,Z 839.06,A -85,B 0,C 180,E1 1216.188,E2 1216.188} C_VEL
LIN {X 0,Y 747.173,Z 839.06,A -85,B 0,C 180,E1 1223.375,E2 1223.375} C_VEL
LIN {X 0,Y 746.97,Z 839.06,A -85,B 0,C 180,E1 1231.528,E2 1231.528} C_VEL
LIN {X 0,Y 746.842,Z 839.06,A -85,B 0,C 180,E1 1239.211,E2 1239.211} C_VEL
LIN {X 0,Y 747.135,Z 839.06,A -85,B 0,C 180,E1 1246.53,E2 1246.53} C_VEL
LIN {X 0,Y 747.067,Z 839.06,A -85,B 0,C 180,E1 1252.448,E2 1252.448} C_VEL
LIN {X 0,Y 746.805,Z 839.06,A -85,B 0,C 180,E1 1260.615,E2 1260.615} C_VEL
LIN {X 0,Y 746.202,Z 839.06,A -85,B 0,C 180,E1 1262.918,E2 1262.918} C_VEL
LIN {X 0,Y 739.014,Z 839.06,A -85,B 0,C 180,E1 1265.6,E2 1265.6} C_VEL
LIN {X 0,Y 739.18,Z 839.06,A -85,B 0,C 180,E1 1274.901,E2 1274.901} C_VEL
LIN {X 0,Y 738.749,Z 839.06,A -85,B 0,C 180,E1 1283.645,E2 1283.645} C_VEL
LIN {X 0,Y 738.64,Z 839.06,A -85,B 0,C 180,E1 1291.467,E2 1291.467} C_VEL
LIN {X 0,Y 738.643,Z 839.06,A -85,B 0,C 180,E1 1298.834,E2 1298.834} C_VEL
LIN {X 0,Y 738.762,Z 839.06,A -85,B 0,C 180,E1 1306.496,E2 1306.496} C_VEL
LIN {X 0,Y 738.97,Z 840.394,A -85,B 0,C 180,E1 1312.283,E2 1312.283} C_VEL
LIN {X 0,Y 743.851,Z 852.305,A -85,B 0,C 180,E1 1312.714,E2 1312.714} C_VEL
LIN {X 0,Y 743.901,Z 942.728,A -85,B 0,C 180,E1 1314.063,E2 1314.063} C_VEL
LIN {X 0,Y 743.054,Z 1013.272,A -85,B 0,C 180,E1 1316.201,E2 1316.201} C_VEL
LIN {X 0,Y 741.783,Z 1084.615,A -85,B 0,C 180,E1 1319.616,E2 1319.616} C_VEL
LIN {X 0,Y 740.449,Z 1149.809,A -85,B 0,C 180,E1 1324.14,E2 1324.14} C_VEL
LIN {X 0,Y 739.487,Z 1201.897,A -85,B 0,C 180,E1 1329.177,E2 1329.177} C_VEL
LIN {X 0,Y 739.082,Z 1238.764,A -85,B 0,C 180,E1 1334.113,E2 1334.113} C_VEL
LIN {X 0,Y 738.963,Z 1265.628,A -85,B 0,C 180,E1 1339.345,E2 1339.345} C_VEL
LIN {X 0,Y 739.086,Z 1281.752,A -85,B 0,C 180,E1 1344.697,E2 1344.697} C_VEL
LIN {X 0,Y 738.939,Z 1286.837,A -85,B 0,C 180,E1 1350.589,E2 1350.589} C_VEL
LIN {X 0,Y 739.152,Z 1280.51,A -85,B 0,C 180,E1 1355.894,E2 1355.894} C_VEL
LIN {X 0,Y 739.17,Z 1260.44,A -85,B 0,C 180,E1 1361.852,E2 1361.852} C_VEL
LIN {X 0,Y 739.5,Z 1229.182,A -85,B 0,C 180,E1 1367.331,E2 1367.331} C_VEL
LIN {X 0,Y 740.209,Z 1183.254,A -85,B 0,C 180,E1 1372.81,E2 1372.81} C_VEL
LIN {X 0,Y 741.157,Z 1123.79,A -85,B 0,C 180,E1 1377.844,E2 1377.844} C_VEL
LIN {X 0,Y 742.319,Z 1055.864,A -85,B 0,C 180,E1 1381.92,E2 1381.92} C_VEL
LIN {X 0,Y 743.438,Z 982.882,A -85,B 0,C 180,E1 1384.855,E2 1384.855} C_VEL
LIN {X 0,Y 744.028,Z 907.956,A -85,B 0,C 180,E1 1386.589,E2 1386.589} C_VEL
LIN {X 0,Y 742.209,Z 846.382,A -85,B 0,C 180,E1 1387.453,E2 1387.453} C_VEL
LIN {X 0,Y 738.783,Z 839.06,A -85,B 0,C 180,E1 1387.812,E2 1387.812} C_VEL
LIN {X 0,Y 738.701,Z 839.06,A -85,B 0,C 180,E1 1396.478,E2 1396.478} C_VEL
LIN {X 0,Y 738.885,Z 839.06,A -85,B 0,C 180,E1 1404.25,E2 1404.25} C_VEL
LIN {X 0,Y 738.886,Z 839.06,A -85,B 0,C 180,E1 1411.11,E2 1411.11} C_VEL
LIN {X 0,Y 738.525,Z 839.06,A -85,B 0,C 180,E1 1417.626,E2 1417.626} C_VEL
LIN {X 0,Y 738.898,Z 839.06,A -85,B 0,C 180,E1 1425.093,E2 1425.093} C_VEL
LIN {X 0,Y 739.195,Z 839.06,A -85,B 0,C 180,E1 1432.299,E2 1432.299} C_VEL
LIN {X 0,Y 738.851,Z 839.06,A -85,B 0,C 180,E1 1440.554,E2 1440.554} C_VEL
LIN {X 0,Y 739.011,Z 839.06,A -85,B 0,C 180,E1 1447.635,E2 1447.635} C_VEL
LIN {X 0,Y 739.316,Z 839.06,A -85,B 0,C 180,E1 1454.829,E2 1454.829} C_VEL
LIN {X 0,Y 738.799,Z 839.06,A -85,B 0,C 180,E1 1463.569,E2 1463.569} C_VEL
LIN {X 0,Y 738.585,Z 839.06,A -85,B 0,C 180,E1 1471.549,E2 1471.549} C_VEL
LIN {X 0,Y 738.713,Z 839.06,A -85,B 0,C 180,E1 1478.743,E2 1478.743} C_VEL
LIN {X 0,Y 738.752,Z 839.06,A -85,B 0,C 180,E1 1486.495,E2 1486.495} C_VEL
LIN {X 0,Y 739.202,Z 840.256,A -85,B 0,C 180,E1 1492.61,E2 1492.61} C_VEL
LIN {X 0,Y 743.969,Z 858.103,A -85,B 0,C 180,E1 1493.101,E2 1493.101} C_VEL
LIN {X 0,Y 743.567,Z 936.272,A -85,B 0,C 180,E1 1494.599,E2 1494.599} C_VEL
LIN {X 0,Y 742.54,Z 1009.58,A -85,B 0,C 180,E1 1497.26,E2 1497.26} C_VEL
LIN {X 0,Y 741.238,Z 1079.443,A -85,B 0,C 180,E1 1501.116,E2 1501.116} C_VEL
LIN {X 0,Y 740.138,Z 1139.851,A -85,B 0,C 180,E1 1505.844,E2 1505.844} C_VEL
LIN {X 0,Y 739.479,Z 1186.943,A -85,B 0,C 180,E1 1510.962,E2 1510.962} C_VEL
LIN {X 0,Y 739.137,Z 1221.805,A -85,B 0,C 180,E1 1516.337,E2 1516.337} C_VEL
LIN {X 0,Y 739.287,Z 1244.308,A -85,B 0,C 180,E1 1521.735,E2 1521.735} C_VEL
LIN {X 0,Y 739.427,Z 1255.391,A -85,B 0,C 180,E1 1527.058,E2 1527.058} C_VEL
LIN {X 0,Y 739.439,Z 1255.313,A -85,B 0,C 180,E1 1532.942,E2 1532.942} C_VEL
LIN {X 0,Y 739.367,Z 1242.071,A -85,B 0,C 180,E1 1538.858,E2 1538.858} C_VEL
LIN {X 0,Y 739.405,Z 1214.551,A -85,B 0,C 180,E1 1544.871,E2 1544.871} C_VEL
LIN {X 0,Y 739.895,Z 1173.572,A -85,B 0,C 180,E1 1550.571,E2 1550.571} C_VEL
LIN {X 0,Y 740.782,Z 1118.984,A -85,B 0,C 180,E1 1555.873,E2 1555.873} C_VEL
LIN {X 0,Y 741.895,Z 1054.193,A -85,B 0,C 180,E1 1560.36,E2 1560.36} C_VEL
LIN {X 0,Y 743.047,Z 982.892,A -85,B 0,C 180,E1 1563.77,E2 1563.77} C_VEL
LIN {X 0,Y 743.922,Z 909.322,A -85,B 0,C 180,E1 1565.967,E2 1565.967} C_VEL
LIN {X 0,Y 742.127,Z 845.206,A -85,B 0,C 180,E1 1567.069,E2 1567.069} C_VEL
LIN {X 0,Y 739.096,Z 839.06,A -85,B 0,C 180,E1 1567.421,E2 1567.421} C_VEL
LIN {X 0,Y 739.327,Z 839.06,A -85,B 0,C 180,E1 1575.106,E2 1575.106} C_VEL
LIN {X 0,Y 738.697,Z 839.06,A -85,B 0,C 180,E1 1584.269,E2 1584.269} C_VEL
LIN {X 0,Y 739.011,Z 839.06,A -85,B 0,C 180,E1 1591.193,E2 1591.193} C_VEL
LIN {X 0,Y 738.842,Z 839.06,A -85,B 0,C 180,E1 1599.211,E2 1599.211} C_VEL
LIN {X 0,Y 738.886,Z 839.06,A -85,B 0,C 180,E1 1607.404,E2 1607.404} C_VEL
LIN {X 0,Y 738.54,Z 839.06,A -85,B 0,C 180,E1 1613.547,E2 1613.547} C_VEL
LIN {X 0,Y 738.797,Z 839.06,A -85,B 0,C 180,E1 1620.622,E2 1620.622} C_VEL
LIN {X 0,Y 739.014,Z 839.06,A -85,B 0,C 180,E1 1625.6,E2 1625.6} C_VEL
LIN {X 0,Y 730.599,Z 839.06,A -85,B 0,C 180,E1 1628.294,E2 1628.294} C_VEL
LIN {X 0,Y 731.064,Z 839.06,A -85,B 0,C 180,E1 1635.071,E2 1635.071} C_VEL
LIN {X 0,Y 731.16,Z 839.06,A -85,B 0,C 180,E1 1642.611,E2 1642.611} C_VEL
LIN {X 0,Y 730.941,Z 839.06,A -85,B 0,C 180,E1 1650.606,E2 1650.606} C_VEL
LIN {X 0,Y 730.66,Z 839.06,A -85,B 0,C 180,E1 1658.818,E2 1658.818} C_VEL
LIN {X 0,Y 730.969,Z 839.06,A -85,B 0,C 180,E1 1665.914,E2 1665.914} C_VEL
LIN {X 0,Y 730.617,Z 840.172,A -85,B 0,C 180,E1 1671.772,E2 1671.772} C_VEL
LIN {X 0,Y 737.45,Z 856.384,A -85,B 0,C 180,E1 1672.384,E2 1672.384} C_VEL
LIN {X 0,Y 737.334,Z 945.051,A -85,B 0,C 180,E1 1673.747,E2 1673.747} C_VEL
LIN {X 0,Y 736.171,Z 1015.582,A -85,B 0,C 180,E1 1675.938,E2 1675.938} C_VEL
LIN {X 0,Y 734.531,Z 1086.57,A -85,B 0,C 180,E1 1679.405,E2 1679.405} C_VEL
LIN {X 0,Y 732.874,Z 1151.586,A -85,B 0,C 180,E1 1684.005,E2 1684.005} C_VEL
LIN {X 0,Y 731.671,Z 1203,A -85,B 0,C 180,E1 1689.074,E2 1689.074} C_VEL
LIN {X 0,Y 731.161,Z 1239.381,A -85,B 0,C 180,E1 1694.032,E2 1694.032} C_VEL
LIN {X 0,Y 731.036,Z 1265.628,A -85,B 0,C 180,E1 1699.228,E2 1699.228} C_VEL
LIN {X 0,Y 731.11,Z 1281.752,A -85,B 0,C 180,E1 1704.639,E2 1704.639} C_VEL
LIN {X 0,Y 730.96,Z 1286.837,A -85,B 0,C 180,E1 1710.595,E2 1710.595} C_VEL
LIN {X 0,Y 731.12,Z 1280.508,A -85,B 0,C 180,E1 1715.96,E2 1715.96} C_VEL
LIN {X 0,Y 731.27,Z 1261.798,A -85,B 0,C 180,E1 1721.678,E2 1721.678} C_VEL
LIN {X 0,Y 731.535,Z 1229.275,A -85,B 0,C 180,E1 1727.513,E2 1727.513} C_VEL
LIN {X 0,Y 732.439,Z 1183.287,A -85,B 0,C 180,E1 1733.063,E2 1733.063} C_VEL
LIN {X 0,Y 733.685,Z 1124.623,A -85,B 0,C 180,E1 1738.092,E2 1738.092} C_VEL
LIN {X 0,Y 735.273,Z 1055.867,A -85,B 0,C 180,E1 1742.263,E2 1742.263} C_VEL
LIN {X 0,Y 736.765,Z 983.456,A -85,B 0,C 180,E1 1745.198,E2 1745.198} C_VEL
LIN {X 0,Y 737.586,Z 908.638,A -85,B 0,C 180,E1 1746.951,E2 1746.951} C_VEL
LIN {X 0,Y 736.053,Z 849.963,A -85,B 0,C 180,E1 1747.777,E2 1747.777} C_VEL
LIN {X 0,Y 730.421,Z 839.06,A -85,B 0,C 180,E1 1748.431,E2 1748.431} C_VEL
LIN {X 0,Y 730.919,Z 839.06,A -85,B 0,C 180,E1 1755.896,E2 1755.896} C_VEL
LIN {X 0,Y 730.954,Z 839.06,A -85,B 0,C 180,E1 1763.69,E2 1763.69} C_VEL
LIN {X 0,Y 731.016,Z 839.06,A -85,B 0,C 180,E1 1770.769,E2 1770.769} C_VEL
LIN {X 0,Y 730.52,Z 839.06,A -85,B 0,C 180,E1 1777.634,E2 1777.634} C_VEL
LIN {X 0,Y 730.944,Z 839.06,A -85,B 0,C 180,E1 1784.967,E2 1784.967} C_VEL
LIN {X 0,Y 731.204,Z 839.06,A -85,B 0,C 180,E1 1792.214,E2 1792.214} C_VEL
LIN {X 0,Y 730.873,Z 839.06,A -85,B 0,C 180,E1 1800.561,E2 1800.561} C_VEL
LIN {X 0,Y 730.954,Z 839.06,A -85,B 0,C 180,E1 1807.719,E2 1807.719} C_VEL
LIN {X 0,Y 731.118,Z 839.06,A -85,B 0,C 180,E1 1815.084,E2 1815.084} C_VEL
LIN {X 0,Y 730.703,Z 839.06,A -85,B 0,C 180,E1 1823.847,E2 1823.847} C_VEL
LIN {X 0,Y 730.99,Z 839.06,A -85,B 0,C 180,E1 1830.525,E2 1830.525} C_VEL
LIN {X 0,Y 730.671,Z 839.06,A -85,B 0,C 180,E1 1838.818,E2 1838.818} C_VEL
LIN {X 0,Y 730.937,Z 839.06,A -85,B 0,C 180,E1 1845.91,E2 1845.91} C_VEL
LIN {X 0,Y 730.941,Z 840.646,A -85,B 0,C 180,E1 1852.119,E2 1852.119} C_VEL
LIN {X 0,Y 737.546,Z 857.712,A -85,B 0,C 180,E1 1852.721,E2 1852.721} C_VEL
LIN {X 0,Y 736.926,Z 935.362,A -85,B 0,C 180,E1 1854.206,E2 1854.206} C_VEL
LIN {X 0,Y 735.59,Z 1010.218,A -85,B 0,C 180,E1 1856.942,E2 1856.942} C_VEL
LIN {X 0,Y 733.923,Z 1079.745,A -85,B 0,C 180,E1 1860.821,E2 1860.821} C_VEL
LIN {X 0,Y 732.487,Z 1139.845,A -85,B 0,C 180,E1 1865.575,E2 1865.575} C_VEL
LIN {X 0,Y 731.633,Z 1187.926,A -85,B 0,C 180,E1 1870.876,E2 1870.876} C_VEL
LIN {X 0,Y 731.233,Z 1221.803,A -85,B 0,C 180,E1 1876.187,E2 1876.187} C_VEL
LIN {X 0,Y 731.007,Z 1246.125,A -85,B 0,C 180,E1 1882.242,E2 1882.242} C_VEL
LIN {X 0,Y 731.43,Z 1255.391,A -85,B 0,C 180,E1 1887.025,E2 1887.025} C_VEL
LIN {X 0,Y 731.414,Z 1255.314,A -85,B 0,C 180,E1 1892.974,E2 1892.974} C_VEL
LIN {X 0,Y 731.316,Z 1242.073,A -85,B 0,C 180,E1 1898.956,E2 1898.956} C_VEL
LIN {X 0,Y 731.438,Z 1214.556,A -85,B 0,C 180,E1 1905.036,E2 1905.036} C_VEL
LIN {X 0,Y 732.059,Z 1173.578,A -85,B 0,C 180,E1 1910.801,E2 1910.801} C_VEL
LIN {X 0,Y 733.196,Z 1119.684,A -85,B 0,C 180,E1 1916.101,E2 1916.101} C_VEL
LIN {X 0,Y 734.709,Z 1054.614,A -85,B 0,C 180,E1 1920.663,E2 1920.663} C_VEL
LIN {X 0,Y 736.195,Z 984.202,A -85,B 0,C 180,E1 1924.073,E2 1924.073} C_VEL
LIN {X 0,Y 737.349,Z 911.012,A -85,B 0,C 180,E1 1926.301,E2 1926.301} C_VEL
LIN {X 0,Y 735.888,Z 849.367,A -85,B 0,C 180,E1 1927.388,E2 1927.388} C_VEL
LIN {X 0,Y 730.827,Z 839.06,A -85,B 0,C 180,E1 1927.832,E2 1927.832} C_VEL
LIN {X 0,Y 730.864,Z 839.06,A -85,B 0,C 180,E1 1935.987,E2 1935.987} C_VEL
LIN {X 0,Y 730.794,Z 839.06,A -85,B 0,C 180,E1 1943.766,E2 1943.766} C_VEL
LIN {X 0,Y 730.682,Z 839.06,A -85,B 0,C 180,E1 1952.007,E2 1952.007} C_VEL
LIN {X 0,Y 730.972,Z 839.06,A -85,B 0,C 180,E1 1958.738,E2 1958.738} C_VEL
LIN {X 0,Y 731.187,Z 839.06,A -85,B 0,C 180,E1 1966.23,E2 1966.23} C_VEL
LIN {X 0,Y 731.114,Z 839.06,A -85,B 0,C 180,E1 1972.282,E2 1972.282} C_VEL
LIN {X 0,Y 730.803,Z 839.06,A -85,B 0,C 180,E1 1980.629,E2 1980.629} C_VEL
LIN {X 0,Y 730.599,Z 839.06,A -85,B 0,C 180,E1 1988.294,E2 1988.294} C_VEL
LIN {X 0,Y 722.156,Z 839.06,A -85,B 0,C 180,E1 1991.005,E2 1991.005} C_VEL
LIN {X 0,Y 722.182,Z 839.06,A -85,B 0,C 180,E1 1996.969,E2 1996.969} C_VEL
LIN {X 0,Y 722.547,Z 839.06,A -85,B 0,C 180,E1 2004.209,E2 2004.209} C_VEL
LIN {X 0,Y 722.496,Z 839.06,A -85,B 0,C 180,E1 2011.681,E2 2011.681} C_VEL
LIN {X 0,Y 722.829,Z 839.06,A -85,B 0,C 180,E1 2018.301,E2 2018.301} C_VEL
LIN {X 0,Y 722.441,Z 839.06,A -85,B 0,C 180,E1 2026.926,E2 2026.926} C_VEL
LIN {X 0,Y 722.381,Z 840.199,A -85,B 0,C 180,E1 2031.255,E2 2031.255} C_VEL
LIN {X 0,Y 731.101,Z 859.469,A -85,B 0,C 180,E1 2032.037,E2 2032.037} C_VEL
LIN {X 0,Y 730.83,Z 945.259,A -85,B 0,C 180,E1 2033.377,E2 2033.377} C_VEL
LIN {X 0,Y 729.338,Z 1016.491,A -85,B 0,C 180,E1 2035.613,E2 2035.613} C_VEL
LIN {X 0,Y 727.307,Z 1087.977,A -85,B 0,C 180,E1 2039.156,E2 2039.156} C_VEL
LIN {X 0,Y 725.297,Z 1153.051,A -85,B 0,C 180,E1 2043.839,E2 2043.839} C_VEL
LIN {X 0,Y 723.835,Z 1204.862,A -85,B 0,C 180,E1 2049.059,E2 2049.059} C_VEL
LIN {X 0,Y 723.181,Z 1241.283,A -85,B 0,C 180,E1 2054.164,E2 2054.164} C_VEL
LIN {X 0,Y 722.971,Z 1266.791,A -85,B 0,C 180,E1 2059.413,E2 2059.413} C_VEL
LIN {X 0,Y 723.142,Z 1281.752,A -85,B 0,C 180,E1 2064.58,E2 2064.58} C_VEL
LIN {X 0,Y 722.955,Z 1286.837,A -85,B 0,C 180,E1 2070.602,E2 2070.602} C_VEL
LIN {X 0,Y 723.109,Z 1280.509,A -85,B 0,C 180,E1 2076.026,E2 2076.026} C_VEL
LIN {X 0,Y 723.26,Z 1262.091,A -85,B 0,C 180,E1 2081.743,E2 2081.743} C_VEL
LIN {X 0,Y 723.591,Z 1229.276,A -85,B 0,C 180,E1 2087.711,E2 2087.711} C_VEL
LIN {X 0,Y 724.674,Z 1181.992,A -85,B 0,C 180,E1 2093.456,E2 2093.456} C_VEL
LIN {X 0,Y 726.336,Z 1121.942,A -85,B 0,C 180,E1 2098.601,E2 2098.601} C_VEL
LIN {X 0,Y 728.371,Z 1053.028,A -85,B 0,C 180,E1 2102.755,E2 2102.755} C_VEL
LIN {X 0,Y 730.13,Z 981.896,A -85,B 0,C 180,E1 2105.618,E2 2105.618} C_VEL
LIN {X 0,Y 731.196,Z 907.476,A -85,B 0,C 180,E1 2107.346,E2 2107.346} C_VEL
LIN {X 0,Y 729.75,Z 853.585,A -85,B 0,C 180,E1 2108.118,E2 2108.118} C_VEL
LIN {X 0,Y 722.197,Z 839.06,A -85,B 0,C 180,E1 2108.943,E2 2108.943} C_VEL
LIN {X 0,Y 722.466,Z 839.06,A -85,B 0,C 180,E1 2116.913,E2 2116.913} C_VEL
LIN {X 0,Y 722.672,Z 839.06,A -85,B 0,C 180,E1 2124.694,E2 2124.694} C_VEL
LIN {X 0,Y 722.749,Z 839.06,A -85,B 0,C 180,E1 2131.776,E2 2131.776} C_VEL
LIN {X 0,Y 722.195,Z 839.06,A -85,B 0,C 180,E1 2138.393,E2 2138.393} C_VEL
LIN {X 0,Y 722.972,Z 839.06,A -85,B 0,C 180,E1 2144.757,E2 2144.757} C_VEL
LIN {X 0,Y 723.229,Z 839.06,A -85,B 0,C 180,E1 2152.128,E2 2152.128} C_VEL
LIN {X 0,Y 722.864,Z 839.06,A -85,B 0,C 180,E1 2160.567,E2 2160.567} C_VEL
LIN {X 0,Y 722.93,Z 839.06,A -85,B 0,C 180,E1 2167.805,E2 2167.805} C_VEL
LIN {X 0,Y 723.069,Z 839.06,A -85,B 0,C 180,E1 2175.17,E2 2175.17} C_VEL
LIN {X 0,Y 722.649,Z 839.06,A -85,B 0,C 180,E1 2183.959,E2 2183.959} C_VEL
LIN {X 0,Y 722.493,Z 839.06,A -85,B 0,C 180,E1 2191.679,E2 2191.679} C_VEL
LIN {X 0,Y 722.884,Z 839.06,A -85,B 0,C 180,E1 2198.21,E2 2198.21} C_VEL
LIN {X 0,Y 722.712,Z 839.06,A -85,B 0,C 180,E1 2206.357,E2 2206.357} C_VEL
LIN {X 0,Y 722.636,Z 840.588,A -85,B 0,C 180,E1 2211.605,E2 2211.605} C_VEL
LIN {X 0,Y 731.176,Z 858.793,A -85,B 0,C 180,E1 2212.354,E2 2212.354} C_VEL
LIN {X 0,Y 730.324,Z 936.539,A -85,B 0,C 180,E1 2213.867,E2 2213.867} C_VEL
LIN {X 0,Y 728.644,Z 1009.738,A -85,B 0,C 180,E1 2216.563,E2 2216.563} C_VEL
LIN {X 0,Y 726.644,Z 1079.286,A -85,B 0,C 180,E1 2220.469,E2 2220.469} C_VEL
LIN {X 0,Y 724.876,Z 1140.477,A -85,B 0,C 180,E1 2225.361,E2 2225.361} C_VEL
LIN {X 0,Y 723.798,Z 1188.328,A -85,B 0,C 180,E1 2230.714,E2 2230.714} C_VEL
LIN {X 0,Y 723.204,Z 1223.516,A -85,B 0,C 180,E1 2236.371,E2 2236.371} C_VEL
LIN {X 0,Y 723.045,Z 1246.124,A -85,B 0,C 180,E1 2242.156,E2 2242.156} C_VEL
LIN {X 0,Y 723.428,Z 1255.391,A -85,B 0,C 180,E1 2246.992,E2 2246.992} C_VEL
LIN {X 0,Y 723.386,Z 1255.314,A -85,B 0,C 180,E1 2253.007,E2 2253.007} C_VEL
LIN {X 0,Y 723.272,Z 1242.075,A -85,B 0,C 180,E1 2259.057,E2 2259.057} C_VEL
LIN {X 0,Y 723.547,Z 1216.327,A -85,B 0,C 180,E1 2264.893,E2 2264.893} C_VEL
LIN {X 0,Y 724.238,Z 1174.784,A -85,B 0,C 180,E1 2270.893,E2 2270.893} C_VEL
LIN {X 0,Y 725.627,Z 1120.85,A -85,B 0,C 180,E1 2276.294,E2 2276.294} C_VEL
LIN {X 0,Y 727.463,Z 1056.645,A -85,B 0,C 180,E1 2280.875,E2 2280.875} C_VEL
LIN {X 0,Y 729.38,Z 985.244,A -85,B 0,C 180,E1 2284.393,E2 2284.393} C_VEL
LIN {X 0,Y 730.856,Z 911.425,A -85,B 0,C 180,E1 2286.666,E2 2286.666} C_VEL
LIN {X 0,Y 729.691,Z 852.999,A -85,B 0,C 180,E1 2287.717,E2 2287.717} C_VEL
LIN {X 0,Y 722.526,Z 839.06,A -85,B 0,C 180,E1 2288.367,E2 2288.367} C_VEL
LIN {X 0,Y 722.669,Z 839.06,A -85,B 0,C 180,E1 2296.447,E2 2296.447} C_VEL
LIN {X 0,Y 722.702,Z 839.06,A -85,B 0,C 180,E1 2303.972,E2 2303.972} C_VEL
LIN {X 0,Y 722.737,Z 839.06,A -85,B 0,C 180,E1 2311.854,E2 2311.854} C_VEL
LIN {X 0,Y 722.548,Z 839.06,A -85,B 0,C 180,E1 2319.766,E2 2319.766} C_VEL
LIN {X 0,Y 722.876,Z 839.06,A -85,B 0,C 180,E1 2327.566,E2 2327.566} C_VEL
LIN {X 0,Y 722.596,Z 839.06,A -85,B 0,C 180,E1 2333.403,E2 2333.403} C_VEL
LIN {X 0,Y 722.795,Z 839.06,A -85,B 0,C 180,E1 2340.636,E2 2340.636} C_VEL
LIN {X 0,Y 722.621,Z 839.06,A -85,B 0,C 180,E1 2348.274,E2 2348.274} C_VEL
LIN {X 0,Y 722.156,Z 839.06,A -85,B 0,C 180,E1 2351.005,E2 2351.005} C_VEL
LIN {X 0,Y 714.913,Z 839.06,A -85,B 0,C 180,E1 2353.778,E2 2353.778} C_VEL
LIN {X 0,Y 714.891,Z 839.06,A -85,B 0,C 180,E1 2363.156,E2 2363.156} C_VEL
LIN {X 0,Y 714.589,Z 839.06,A -85,B 0,C 180,E1 2371.385,E2 2371.385} C_VEL
LIN {X 0,Y 714.489,Z 839.06,A -85,B 0,C 180,E1 2379.147,E2 2379.147} C_VEL
LIN {X 0,Y 714.678,Z 839.06,A -85,B 0,C 180,E1 2386.342,E2 2386.342} C_VEL
LIN {X 0,Y 714.173,Z 840.153,A -85,B 0,C 180,E1 2390.724,E2 2390.724} C_VEL
LIN {X 0,Y 724.788,Z 862.241,A -85,B 0,C 180,E1 2391.681,E2 2391.681} C_VEL
LIN {X 0,Y 724.325,Z 946.94,A -85,B 0,C 180,E1 2393.035,E2 2393.035} C_VEL
LIN {X 0,Y 722.482,Z 1018.675,A -85,B 0,C 180,E1 2395.334,E2 2395.334} C_VEL
LIN {X 0,Y 720.1,Z 1089.377,A -85,B 0,C 180,E1 2398.902,E2 2398.902} C_VEL
LIN {X 0,Y 717.747,Z 1153.352,A -85,B 0,C 180,E1 2403.569,E2 2403.569} C_VEL
LIN {X 0,Y 716.084,Z 1204.864,A -85,B 0,C 180,E1 2408.821,E2 2408.821} C_VEL
LIN {X 0,Y 715.297,Z 1241.284,A -85,B 0,C 180,E1 2413.984,E2 2413.984} C_VEL
LIN {X 0,Y 715.036,Z 1266.792,A -85,B 0,C 180,E1 2419.294,E2 2419.294} C_VEL
LIN {X 0,Y 715.166,Z 1281.752,A -85,B 0,C 180,E1 2424.519,E2 2424.519} C_VEL
LIN {X 0,Y 714.958,Z 1286.837,A -85,B 0,C 180,E1 2430.609,E2 2430.609} C_VEL
LIN {X 0,Y 715.106,Z 1280.509,A -85,B 0,C 180,E1 2436.094,E2 2436.094} C_VEL
LIN {X 0,Y 715.356,Z 1263.155,A -85,B 0,C 180,E1 2441.631,E2 2441.631} C_VEL
LIN {X 0,Y 715.706,Z 1230.799,A -85,B 0,C 180,E1 2447.69,E2 2447.69} C_VEL
LIN {X 0,Y 716.969,Z 1185.212,A -85,B 0,C 180,E1 2453.392,E2 2453.392} C_VEL
LIN {X 0,Y 718.858,Z 1127.588,A -85,B 0,C 180,E1 2458.502,E2 2458.502} C_VEL
LIN {X 0,Y 721.154,Z 1060.303,A -85,B 0,C 180,E1 2462.739,E2 2462.739} C_VEL
LIN {X 0,Y 723.399,Z 987.635,A -85,B 0,C 180,E1 2465.809,E2 2465.809} C_VEL
LIN {X 0,Y 724.752,Z 912.452,A -85,B 0,C 180,E1 2467.658,E2 2467.658} C_VEL
LIN {X 0,Y 723.14,Z 856.054,A -85,B 0,C 180,E1 2468.499,E2 2468.499} C_VEL
LIN {X 0,Y 714.045,Z 839.06,A -85,B 0,C 180,E1 2469.435,E2 2469.435} C_VEL
LIN {X 0,Y 714.668,Z 839.06,A -85,B 0,C 180,E1 2476.325,E2 2476.325} C_VEL
LIN {X 0,Y 714.625,Z 839.06,A -85,B 0,C 180,E1 2484.873,E2 2484.873} C_VEL
LIN {X 0,Y 714.764,Z 839.06,A -85,B 0,C 180,E1 2491.817,E2 2491.817} C_VEL
LIN {X 0,Y 714.268,Z 839.06,A -85,B 0,C 180,E1 2498.141,E2 2498.141} C_VEL
LIN {X 0,Y 714.802,Z 839.06,A -85,B 0,C 180,E1 2505.094,E2 2505.094} C_VEL
LIN {X 0,Y 715.225,Z 839.06,A -85,B 0,C 180,E1 2512.039,E2 2512.039} C_VEL
LIN {X 0,Y 714.867,Z 839.06,A -85,B 0,C 180,E1 2520.573,E2 2520.573} C_VEL
LIN {X 0,Y 714.876,Z 839.06,A -85,B 0,C 180,E1 2527.894,E2 2527.894} C_VEL
LIN {X 0,Y 714.96,Z 839.06,A -85,B 0,C 180,E1 2535.346,E2 2535.346} C_VEL
LIN {X 0,Y 714.928,Z 839.06,A -85,B 0,C 180,E1 2543.078,E2 2543.078} C_VEL
LIN {X 0,Y 714.618,Z 839.06,A -85,B 0,C 180,E1 2551.302,E2 2551.302} C_VEL
LIN {X 0,Y 714.484,Z 839.06,A -85,B 0,C 180,E1 2559.145,E2 2559.145} C_VEL
LIN {X 0,Y 714.421,Z 839.06,A -85,B 0,C 180,E1 2567.059,E2 2567.059} C_VEL
LIN {X 0,Y 714.36,Z 840.448,A -85,B 0,C 180,E1 2571.076,E2 2571.076} C_VEL
LIN {X 0,Y 724.874,Z 862.811,A -85,B 0,C 180,E1 2572.019,E2 2572.019} C_VEL
LIN {X 0,Y 723.747,Z 940.041,A -85,B 0,C 180,E1 2573.59,E2 2573.59} C_VEL
LIN {X 0,Y 721.689,Z 1013.131,A -85,B 0,C 180,E1 2576.361,E2 2576.361} C_VEL
LIN {X 0,Y 719.248,Z 1082.911,A -85,B 0,C 180,E1 2580.386,E2 2580.386} C_VEL
LIN {X 0,Y 717.129,Z 1144.01,A -85,B 0,C 180,E1 2585.419,E2 2585.419} C_VEL
LIN {X 0,Y 715.776,Z 1191.852,A -85,B 0,C 180,E1 2590.968,E2 2590.968} C_VEL
LIN {X 0,Y 715.17,Z 1224.917,A -85,B 0,C 180,E1 2596.496,E2 2596.496} C_VEL
LIN {X 0,Y 715.085,Z 1246.123,A -85,B 0,C 180,E1 2602.068,E2 2602.068} C_VEL
LIN {X 0,Y 715.424,Z 1255.39,A -85,B 0,C 180,E1 2606.959,E2 2606.959} C_VEL
LIN {X 0,Y 715.359,Z 1255.314,A -85,B 0,C 180,E1 2613.041,E2 2613.041} C_VEL
LIN {X 0,Y 715.236,Z 1242.078,A -85,B 0,C 180,E1 2619.16,E2 2619.16} C_VEL
LIN {X 0,Y 715.577,Z 1216.424,A -85,B 0,C 180,E1 2625.047,E2 2625.047} C_VEL
LIN {X 0,Y 716.405,Z 1175.32,A -85,B 0,C 180,E1 2631.069,E2 2631.069} C_VEL
LIN {X 0,Y 718.04,Z 1121.458,A -85,B 0,C 180,E1 2636.54,E2 2636.54} C_VEL
LIN {X 0,Y 720.32,Z 1056.538,A -85,B 0,C 180,E1 2641.223,E2 2641.223} C_VEL
LIN {X 0,Y 722.564,Z 986.624,A -85,B 0,C 180,E1 2644.705,E2 2644.705} C_VEL
LIN {X 0,Y 724.355,Z 912.743,A -85,B 0,C 180,E1 2647.019,E2 2647.019} C_VEL
LIN {X 0,Y 723.349,Z 855.943,A -85,B 0,C 180,E1 2648.07,E2 2648.07} C_VEL
LIN {X 0,Y 714.216,Z 839.06,A -85,B 0,C 180,E1 2649.019,E2 2649.019} C_VEL
LIN {X 0,Y 714.68,Z 839.06,A -85,B 0,C 180,E1 2656.423,E2 2656.423} C_VEL
LIN {X 0,Y 714.6,Z 839.06,A -85,B 0,C 180,E1 2664.32,E2 2664.32} C_VEL
LIN {X 0,Y 714.755,Z 839.06,A -85,B 0,C 180,E1 2671.817,E2 2671.817} C_VEL
LIN {X 0,Y 714.632,Z 839.06,A -85,B 0,C 180,E1 2679.532,E2 2679.532} C_VEL
LIN {X 0,Y 714.944,Z 839.06,A -85,B 0,C 180,E1 2687.161,E2 2687.161} C_VEL
LIN {X 0,Y 714.619,Z 839.06,A -85,B 0,C 180,E1 2693.33,E2 2693.33} C_VEL
LIN {X 0,Y 714.801,Z 839.06,A -85,B 0,C 180,E1 2700.643,E2 2700.643} C_VEL
LIN {X 0,Y 714.755,Z 839.06,A -85,B 0,C 180,E1 2707.966,E2 2707.966} C_VEL
LIN {X 0,Y 714.913,Z 839.06,A -85,B 0,C 180,E1 2713.778,E2 2713.778} C_VEL
LIN {X 0,Y 706.324,Z 839.06,A -85,B 0,C 180,E1 2716.569,E2 2716.569} C_VEL
LIN {X 0,Y 706.552,Z 839.06,A -85,B 0,C 180,E1 2724.054,E2 2724.054} C_VEL
LIN {X 0,Y 706.421,Z 839.06,A -85,B 0,C 180,E1 2731.912,E2 2731.912} C_VEL
LIN {X 0,Y 706.411,Z 839.06,A -85,B 0,C 180,E1 2739.361,E2 2739.361} C_VEL
LIN {X 0,Y 706.751,Z 839.06,A -85,B 0,C 180,E1 2746.035,E2 2746.035} C_VEL
LIN {X 0,Y 706.189,Z 840.782,A -85,B 0,C 180,E1 2750.201,E2 2750.201} C_VEL
LIN {X 0,Y 718.526,Z 864.229,A -85,B 0,C 180,E1 2751.31,E2 2751.31} C_VEL
LIN {X 0,Y 717.83,Z 948.69,A -85,B 0,C 180,E1 2752.688,E2 2752.688} C_VEL
LIN {X 0,Y 715.663,Z 1020.367,A -85,B 0,C 180,E1 2755.029,E2 2755.029} C_VEL
LIN {X 0,Y 712.844,Z 1091.952,A -85,B 0,C 180,E1 2758.716,E2 2758.716} C_VEL
LIN {X 0,Y 710.141,Z 1156.433,A -85,B 0,C 180,E1 2763.538,E2 2763.538} C_VEL
LIN {X 0,Y 708.233,Z 1206.911,A -85,B 0,C 180,E1 2768.825,E2 2768.825} C_VEL
LIN {X 0,Y 707.297,Z 1243.052,A -85,B 0,C 180,E1 2774.118,E2 2774.118} C_VEL
LIN {X 0,Y 706.978,Z 1267.954,A -85,B 0,C 180,E1 2779.484,E2 2779.484} C_VEL
LIN {X 0,Y 706.926,Z 1282.875,A -85,B 0,C 180,E1 2785.073,E2 2785.073} C_VEL
LIN {X 0,Y 706.953,Z 1286.837,A -85,B 0,C 180,E1 2790.616,E2 2790.616} C_VEL
LIN {X 0,Y 707.101,Z 1280.509,A -85,B 0,C 180,E1 2796.163,E2 2796.163} C_VEL
LIN {X 0,Y 707.179,Z 1261.906,A -85,B 0,C 180,E1 2802.058,E2 2802.058} C_VEL
LIN {X 0,Y 707.737,Z 1230.815,A -85,B 0,C 180,E1 2807.893,E2 2807.893} C_VEL
LIN {X 0,Y 709.247,Z 1185.469,A -85,B 0,C 180,E1 2813.635,E2 2813.635} C_VEL
LIN {X 0,Y 711.478,Z 1127.589,A -85,B 0,C 180,E1 2818.826,E2 2818.826} C_VEL
LIN {X 0,Y 714.159,Z 1060.571,A -85,B 0,C 180,E1 2823.086,E2 2823.086} C_VEL
LIN {X 0,Y 716.794,Z 987.638,A -85,B 0,C 180,E1 2826.191,E2 2826.191} C_VEL
LIN {X 0,Y 718.395,Z 913.416,A -85,B 0,C 180,E1 2828.033,E2 2828.033} C_VEL
LIN {X 0,Y 716.949,Z 859.688,A -85,B 0,C 180,E1 2828.848,E2 2828.848} C_VEL
LIN {X 0,Y 705.959,Z 839.06,A -85,B 0,C 180,E1 2829.949,E2 2829.949} C_VEL
LIN {X 0,Y 706.736,Z 839.06,A -85,B 0,C 180,E1 2836.022,E2 2836.022} C_VEL
LIN {X 0,Y 706.791,Z 839.06,A -85,B 0,C 180,E1 2843.777,E2 2843.777} C_VEL
LIN {X 0,Y 706.839,Z 839.06,A -85,B 0,C 180,E1 2851.081,E2 2851.081} C_VEL
LIN {X 0,Y 706.356,Z 839.06,A -85,B 0,C 180,E1 2857.883,E2 2857.883} C_VEL
LIN {X 0,Y 706.554,Z 839.06,A -85,B 0,C 180,E1 2865.667,E2 2865.667} C_VEL
LIN {X 0,Y 706.708,Z 839.06,A -85,B 0,C 180,E1 2873.183,E2 2873.183} C_VEL
LIN {X 0,Y 706.858,Z 839.06,A -85,B 0,C 180,E1 2880.58,E2 2880.58} C_VEL
LIN {X 0,Y 706.826,Z 839.06,A -85,B 0,C 180,E1 2887.984,E2 2887.984} C_VEL
LIN {X 0,Y 706.842,Z 839.06,A -85,B 0,C 180,E1 2895.527,E2 2895.527} C_VEL
LIN {X 0,Y 706.573,Z 839.06,A -85,B 0,C 180,E1 2904.056,E2 2904.056} C_VEL
LIN {X 0,Y 706.395,Z 839.06,A -85,B 0,C 180,E1 2911.907,E2 2911.907} C_VEL
LIN {X 0,Y 706.47,Z 839.06,A -85,B 0,C 180,E1 2919.265,E2 2919.265} C_VEL
LIN {X 0,Y 706.805,Z 839.06,A -85,B 0,C 180,E1 2925.929,E2 2925.929} C_VEL
LIN {X 0,Y 706.166,Z 840.112,A -85,B 0,C 180,E1 2930.534,E2 2930.534} C_VEL
LIN {X 0,Y 718.548,Z 864.309,A -85,B 0,C 180,E1 2931.645,E2 2931.645} C_VEL
LIN {X 0,Y 717.194,Z 942.054,A -85,B 0,C 180,E1 2933.265,E2 2933.265} C_VEL
LIN {X 0,Y 714.733,Z 1015.699,A -85,B 0,C 180,E1 2936.115,E2 2936.115} C_VEL
LIN {X 0,Y 711.878,Z 1085.639,A -85,B 0,C 180,E1 2940.24,E2 2940.24} C_VEL
LIN {X 0,Y 709.413,Z 1145.947,A -85,B 0,C 180,E1 2945.336,E2 2945.336} C_VEL
LIN {X 0,Y 707.911,Z 1192.955,A -85,B 0,C 180,E1 2950.911,E2 2950.911} C_VEL
LIN {X 0,Y 707.138,Z 1226.464,A -85,B 0,C 180,E1 2956.656,E2 2956.656} C_VEL
LIN {X 0,Y 707.153,Z 1246.121,A -85,B 0,C 180,E1 2961.978,E2 2961.978} C_VEL
LIN {X 0,Y 707.421,Z 1255.39,A -85,B 0,C 180,E1 2966.924,E2 2966.924} C_VEL
LIN {X 0,Y 707.332,Z 1255.314,A -85,B 0,C 180,E1 2973.075,E2 2973.075} C_VEL
LIN {X 0,Y 707.23,Z 1242.08,A -85,B 0,C 180,E1 2979.264,E2 2979.264} C_VEL
LIN {X 0,Y 707.586,Z 1216.495,A -85,B 0,C 180,E1 2985.209,E2 2985.209} C_VEL
LIN {X 0,Y 708.565,Z 1176.29,A -85,B 0,C 180,E1 2991.196,E2 2991.196} C_VEL
LIN {X 0,Y 710.484,Z 1121.9,A -85,B 0,C 180,E1 2996.806,E2 2996.806} C_VEL
LIN {X 0,Y 713.13,Z 1057.614,A -85,B 0,C 180,E1 3001.505,E2 3001.505} C_VEL
LIN {X 0,Y 715.823,Z 987.44,A -85,B 0,C 180,E1 3005.045,E2 3005.045} C_VEL
LIN {X 0,Y 717.889,Z 913.91,A -85,B 0,C 180,E1 3007.381,E2 3007.381} C_VEL
LIN {X 0,Y 717.12,Z 859.549,A -85,B 0,C 180,E1 3008.417,E2 3008.417} C_VEL
LIN {X 0,Y 706.06,Z 839.06,A -85,B 0,C 180,E1 3009.558,E2 3009.558} C_VEL
LIN {X 0,Y 706.775,Z 839.06,A -85,B 0,C 180,E1 3016.018,E2 3016.018} C_VEL
LIN {X 0,Y 706.64,Z 839.06,A -85,B 0,C 180,E1 3023.856,E2 3023.856} C_VEL
LIN {X 0,Y 706.812,Z 839.06,A -85,B 0,C 180,E1 3031.161,E2 3031.161} C_VEL
LIN {X 0,Y 706.67,Z 839.06,A -85,B 0,C 180,E1 3039.29,E2 3039.29} C_VEL
LIN {X 0,Y 706.958,Z 839.06,A -85,B 0,C 180,E1 3047.013,E2 3047.013} C_VEL
LIN {X 0,Y 706.641,Z 839.06,A -85,B 0,C 180,E1 3053.254,E2 3053.254} C_VEL
LIN {X 0,Y 706.793,Z 839.06,A -85,B 0,C 180,E1 3060.65,E2 3060.65} C_VEL
LIN {X 0,Y 706.712,Z 839.06,A -85,B 0,C 180,E1 3068.057,E2 3068.057} C_VEL
LIN {X 0,Y 706.74,Z 839.06,A -85,B 0,C 180,E1 3075.602,E2 3075.602} C_VEL
LIN {X 0,Y 706.324,Z 839.06,A -85,B 0,C 180,E1 3076.569,E2 3076.569} C_VEL
LIN {X 0,Y 698.182,Z 839.06,A -85,B 0,C 180,E1 3079.392,E2 3079.392} C_VEL
LIN {X 0,Y 698.314,Z 839.06,A -85,B 0,C 180,E1 3086.488,E2 3086.488} C_VEL
LIN {X 0,Y 698.205,Z 839.06,A -85,B 0,C 180,E1 3093.692,E2 3093.692} C_VEL
LIN {X 0,Y 698.282,Z 839.06,A -85,B 0,C 180,E1 3099.91,E2 3099.91} C_VEL
LIN {X 0,Y 698.435,Z 839.06,A -85,B 0,C 180,E1 3106.79,E2 3106.79} C_VEL
LIN {X 0,Y 698.046,Z 840.276,A -85,B 0,C 180,E1 3109.635,E2 3109.635} C_VEL
LIN {X 0,Y 712.261,Z 867.523,A -85,B 0,C 180,E1 3110.948,E2 3110.948} C_VEL
LIN {X 0,Y 711.37,Z 950.31,A -85,B 0,C 180,E1 3112.332,E2 3112.332} C_VEL
LIN {X 0,Y 708.912,Z 1021.052,A -85,B 0,C 180,E1 3114.677,E2 3114.677} C_VEL
LIN {X 0,Y 705.751,Z 1091.564,A -85,B 0,C 180,E1 3118.34,E2 3118.34} C_VEL
LIN {X 0,Y 702.658,Z 1155.969,A -85,B 0,C 180,E1 3123.192,E2 3123.192} C_VEL
LIN {X 0,Y 700.493,Z 1206.913,A -85,B 0,C 180,E1 3128.579,E2 3128.579} C_VEL
LIN {X 0,Y 699.424,Z 1243.054,A -85,B 0,C 180,E1 3133.935,E2 3133.935} C_VEL
LIN {X 0,Y 699.035,Z 1267.955,A -85,B 0,C 180,E1 3139.363,E2 3139.363} C_VEL
LIN {X 0,Y 698.969,Z 1282.874,A -85,B 0,C 180,E1 3145.016,E2 3145.016} C_VEL
LIN {X 0,Y 698.964,Z 1286.837,A -85,B 0,C 180,E1 3150.623,E2 3150.623} C_VEL
LIN {X 0,Y 699.084,Z 1280.509,A -85,B 0,C 180,E1 3156.234,E2 3156.234} C_VEL
LIN {X 0,Y 699.195,Z 1261.907,A -85,B 0,C 180,E1 3162.198,E2 3162.198} C_VEL
LIN {X 0,Y 699.843,Z 1230.517,A -85,B 0,C 180,E1 3168.146,E2 3168.146} C_VEL
LIN {X 0,Y 701.528,Z 1184.425,A -85,B 0,C 180,E1 3174.022,E2 3174.022} C_VEL
LIN {X 0,Y 704.157,Z 1126.199,A -85,B 0,C 180,E1 3179.261,E2 3179.261} C_VEL
LIN {X 0,Y 707.322,Z 1058.591,A -85,B 0,C 180,E1 3183.556,E2 3183.556} C_VEL
LIN {X 0,Y 710.237,Z 986.731,A -85,B 0,C 180,E1 3186.61,E2 3186.61} C_VEL
LIN {X 0,Y 712.109,Z 912.786,A -85,B 0,C 180,E1 3188.441,E2 3188.441} C_VEL
LIN {X 0,Y 710.799,Z 863.154,A -85,B 0,C 180,E1 3189.204,E2 3189.204} C_VEL
LIN {X 0,Y 697.924,Z 839.06,A -85,B 0,C 180,E1 3190.57,E2 3190.57} C_VEL
LIN {X 0,Y 698.467,Z 839.06,A -85,B 0,C 180,E1 3196.776,E2 3196.776} C_VEL
LIN {X 0,Y 698.592,Z 839.06,A -85,B 0,C 180,E1 3204.82,E2 3204.82} C_VEL
LIN {X 0,Y 698.689,Z 839.06,A -85,B 0,C 180,E1 3212.128,E2 3212.128} C_VEL
LIN {X 0,Y 698.077,Z 839.06,A -85,B 0,C 180,E1 3218.947,E2 3218.947} C_VEL
LIN {X 0,Y 698.59,Z 839.06,A -85,B 0,C 180,E1 3225.5,E2 3225.5} C_VEL
LIN {X 0,Y 698.729,Z 839.06,A -85,B 0,C 180,E1 3233.105,E2 3233.105} C_VEL
LIN {X 0,Y 698.848,Z 839.06,A -85,B 0,C 180,E1 3240.586,E2 3240.586} C_VEL
LIN {X 0,Y 698.567,Z 839.06,A -85,B 0,C 180,E1 3248.581,E2 3248.581} C_VEL
LIN {X 0,Y 698.732,Z 839.06,A -85,B 0,C 180,E1 3255.712,E2 3255.712} C_VEL
LIN {X 0,Y 698.716,Z 839.06,A -85,B 0,C 180,E1 3263.646,E2 3263.646} C_VEL
LIN {X 0,Y 698.641,Z 839.06,A -85,B 0,C 180,E1 3270.871,E2 3270.871} C_VEL
LIN {X 0,Y 698.409,Z 839.06,A -85,B 0,C 180,E1 3279.497,E2 3279.497} C_VEL
LIN {X 0,Y 698.446,Z 839.06,A -85,B 0,C 180,E1 3286.79,E2 3286.79} C_VEL
LIN {X 0,Y 698.13,Z 840.571,A -85,B 0,C 180,E1 3289.995,E2 3289.995} C_VEL
LIN {X 0,Y 712.31,Z 868.872,A -85,B 0,C 180,E1 3291.311,E2 3291.311} C_VEL
LIN {X 0,Y 710.55,Z 944.961,A -85,B 0,C 180,E1 3292.961,E2 3292.961} C_VEL
LIN {X 0,Y 707.738,Z 1019.033,A -85,B 0,C 180,E1 3295.902,E2 3295.902} C_VEL
LIN {X 0,Y 704.504,Z 1087.896,A -85,B 0,C 180,E1 3300.069,E2 3300.069} C_VEL
LIN {X 0,Y 701.719,Z 1147.735,A -85,B 0,C 180,E1 3305.236,E2 3305.236} C_VEL
LIN {X 0,Y 700.047,Z 1194.059,A -85,B 0,C 180,E1 3310.852,E2 3310.852} C_VEL
LIN {X 0,Y 699.226,Z 1226.46,A -85,B 0,C 180,E1 3316.502,E2 3316.502} C_VEL
LIN {X 0,Y 698.952,Z 1247.752,A -85,B 0,C 180,E1 3322.512,E2 3322.512} C_VEL
LIN {X 0,Y 698.866,Z 1256.414,A -85,B 0,C 180,E1 3328.132,E2 3328.132} C_VEL
LIN {X 0,Y 699.338,Z 1255.315,A -85,B 0,C 180,E1 3333.111,E2 3333.111} C_VEL
LIN {X 0,Y 699.196,Z 1242.082,A -85,B 0,C 180,E1 3339.372,E2 3339.372} C_VEL
LIN {X 0,Y 699.547,Z 1215.95,A -85,B 0,C 180,E1 3345.488,E2 3345.488} C_VEL
LIN {X 0,Y 700.728,Z 1176.513,A -85,B 0,C 180,E1 3351.418,E2 3351.418} C_VEL
LIN {X 0,Y 702.955,Z 1123.239,A -85,B 0,C 180,E1 3356.997,E2 3356.997} C_VEL
LIN {X 0,Y 705.95,Z 1058.689,A -85,B 0,C 180,E1 3361.793,E2 3361.793} C_VEL
LIN {X 0,Y 709.067,Z 988.509,A -85,B 0,C 180,E1 3365.382,E2 3365.382} C_VEL
LIN {X 0,Y 711.436,Z 915.812,A -85,B 0,C 180,E1 3367.733,E2 3367.733} C_VEL
LIN {X 0,Y 710.934,Z 862.936,A -85,B 0,C 180,E1 3368.771,E2 3368.771} C_VEL
LIN {X 0,Y 697.948,Z 839.06,A -85,B 0,C 180,E1 3370.146,E2 3370.146} C_VEL
LIN {X 0,Y 698.468,Z 839.06,A -85,B 0,C 180,E1 3376.874,E2 3376.874} C_VEL
LIN {X 0,Y 698.373,Z 839.06,A -85,B 0,C 180,E1 3384.895,E2 3384.895} C_VEL
LIN {X 0,Y 698.526,Z 839.06,A -85,B 0,C 180,E1 3392.202,E2 3392.202} C_VEL
LIN {X 0,Y 698.736,Z 839.06,A -85,B 0,C 180,E1 3399.044,E2 3399.044} C_VEL
LIN {X 0,Y 698.966,Z 839.06,A -85,B 0,C 180,E1 3406.862,E2 3406.862} C_VEL
LIN {X 0,Y 698.664,Z 839.06,A -85,B 0,C 180,E1 3413.176,E2 3413.176} C_VEL
LIN {X 0,Y 698.787,Z 839.06,A -85,B 0,C 180,E1 3420.658,E2 3420.658} C_VEL
LIN {X 0,Y 698.508,Z 839.06,A -85,B 0,C 180,E1 3428.553,E2 3428.553} C_VEL
LIN {X 0,Y 698.659,Z 839.06,A -85,B 0,C 180,E1 3435.788,E2 3435.788} C_VEL
LIN {X 0,Y 698.182,Z 839.06,A -85,B 0,C 180,E1 3439.392,E2 3439.392} C_VEL
LIN {X 0,Y 690.789,Z 839.06,A -85,B 0,C 180,E1 3442.269,E2 3442.269} C_VEL
LIN {X 0,Y 690.553,Z 839.06,A -85,B 0,C 180,E1 3451.127,E2 3451.127} C_VEL
LIN {X 0,Y 690.508,Z 839.06,A -85,B 0,C 180,E1 3458.817,E2 3458.817} C_VEL
LIN {X 0,Y 690.514,Z 839.06,A -85,B 0,C 180,E1 3466.169,E2 3466.169} C_VEL
LIN {X 0,Y 690.06,Z 840.263,A -85,B 0,C 180,E1 3469.069,E2 3469.069} C_VEL
LIN {X 0,Y 706.019,Z 871.766,A -85,B 0,C 180,E1 3470.59,E2 3470.59} C_VEL
LIN {X 0,Y 704.954,Z 952.322,A -85,B 0,C 180,E1 3471.981,E2 3471.981} C_VEL
LIN {X 0,Y 702.148,Z 1023.114,A -85,B 0,C 180,E1 3474.377,E2 3474.377} C_VEL
LIN {X 0,Y 698.531,Z 1094.055,A -85,B 0,C 180,E1 3478.139,E2 3478.139} C_VEL
LIN {X 0,Y 695.095,Z 1158.139,A -85,B 0,C 180,E1 3483.074,E2 3483.074} C_VEL
LIN {X 0,Y 692.693,Z 1208.002,A -85,B 0,C 180,E1 3488.464,E2 3488.464} C_VEL
LIN {X 0,Y 691.576,Z 1243.056,A -85,B 0,C 180,E1 3493.747,E2 3493.747} C_VEL
LIN {X 0,Y 691.007,Z 1269.114,A -85,B 0,C 180,E1 3499.558,E2 3499.558} C_VEL
LIN {X 0,Y 690.988,Z 1282.874,A -85,B 0,C 180,E1 3504.959,E2 3504.959} C_VEL
LIN {X 0,Y 690.857,Z 1286.743,A -85,B 0,C 180,E1 3510.977,E2 3510.977} C_VEL
LIN {X 0,Y 691.047,Z 1280.509,A -85,B 0,C 180,E1 3516.307,E2 3516.307} C_VEL
LIN {X 0,Y 691.225,Z 1262.451,A -85,B 0,C 180,E1 3522.212,E2 3522.212} C_VEL
LIN {X 0,Y 691.933,Z 1231.315,A -85,B 0,C 180,E1 3528.239,E2 3528.239} C_VEL
LIN {X 0,Y 693.827,Z 1186.261,A -85,B 0,C 180,E1 3534.108,E2 3534.108} C_VEL
LIN {X 0,Y 696.776,Z 1127.63,A -85,B 0,C 180,E1 3539.49,E2 3539.49} C_VEL
LIN {X 0,Y 700.364,Z 1059.838,A -85,B 0,C 180,E1 3543.865,E2 3543.865} C_VEL
LIN {X 0,Y 703.658,Z 988.639,A -85,B 0,C 180,E1 3546.943,E2 3546.943} C_VEL
LIN {X 0,Y 705.799,Z 913.745,A -85,B 0,C 180,E1 3548.831,E2 3548.831} C_VEL
LIN {X 0,Y 704.481,Z 866.042,A -85,B 0,C 180,E1 3549.587,E2 3549.587} C_VEL
LIN {X 0,Y 689.967,Z 839.06,A -85,B 0,C 180,E1 3551.048,E2 3551.048} C_VEL
LIN {X 0,Y 690.226,Z 839.06,A -85,B 0,C 180,E1 3557.852,E2 3557.852} C_VEL
LIN {X 0,Y 690.512,Z 839.06,A -85,B 0,C 180,E1 3565.881,E2 3565.881} C_VEL
LIN {X 0,Y 690.703,Z 839.06,A -85,B 0,C 180,E1 3573.197,E2 3573.197} C_VEL
LIN {X 0,Y 690.252,Z 839.06,A -85,B 0,C 180,E1 3581.377,E2 3581.377} C_VEL
LIN {X 0,Y 690.208,Z 839.06,A -85,B 0,C 180,E1 3588.178,E2 3588.178} C_VEL
LIN {X 0,Y 690.361,Z 839.06,A -85,B 0,C 180,E1 3594.288,E2 3594.288} C_VEL
LIN {X 0,Y 690.802,Z 839.06,A -85,B 0,C 180,E1 3600.72,E2 3600.72} C_VEL
LIN {X 0,Y 690.74,Z 839.06,A -85,B 0,C 180,E1 3608.172,E2 3608.172} C_VEL
LIN {X 0,Y 690.632,Z 839.06,A -85,B 0,C 180,E1 3615.901,E2 3615.901} C_VEL
LIN {X 0,Y 690.565,Z 839.06,A -85,B 0,C 180,E1 3624.171,E2 3624.171} C_VEL
LIN {X 0,Y 690.354,Z 839.06,A -85,B 0,C 180,E1 3632.152,E2 3632.152} C_VEL
LIN {X 0,Y 690.554,Z 839.06,A -85,B 0,C 180,E1 3638.721,E2 3638.721} C_VEL
LIN {X 0,Y 690.549,Z 839.06,A -85,B 0,C 180,E1 3646.171,E2 3646.171} C_VEL
LIN {X 0,Y 690.017,Z 840.285,A -85,B 0,C 180,E1 3649.425,E2 3649.425} C_VEL
LIN {X 0,Y 706.022,Z 871.482,A -85,B 0,C 180,E1 3650.942,E2 3650.942} C_VEL
LIN {X 0,Y 703.982,Z 947.151,A -85,B 0,C 180,E1 3652.633,E2 3652.633} C_VEL
LIN {X 0,Y 700.782,Z 1021.075,A -85,B 0,C 180,E1 3655.63,E2 3655.63} C_VEL
LIN {X 0,Y 697.144,Z 1089.583,A -85,B 0,C 180,E1 3659.853,E2 3659.853} C_VEL
LIN {X 0,Y 694.037,Z 1149.65,A -85,B 0,C 180,E1 3665.148,E2 3665.148} C_VEL
LIN {X 0,Y 692.155,Z 1195.497,A -85,B 0,C 180,E1 3670.842,E2 3670.842} C_VEL
LIN {X 0,Y 691.2,Z 1227.922,A -85,B 0,C 180,E1 3676.666,E2 3676.666} C_VEL
LIN {X 0,Y 691.006,Z 1247.747,A -85,B 0,C 180,E1 3682.425,E2 3682.425} C_VEL
LIN {X 0,Y 690.871,Z 1256.414,A -85,B 0,C 180,E1 3688.111,E2 3688.111} C_VEL
LIN {X 0,Y 691.161,Z 1254.964,A -85,B 0,C 180,E1 3693.483,E2 3693.483} C_VEL
LIN {X 0,Y 691.154,Z 1242.084,A -85,B 0,C 180,E1 3699.482,E2 3699.482} C_VEL
LIN {X 0,Y 691.622,Z 1216.95,A -85,B 0,C 180,E1 3705.486,E2 3705.486} C_VEL
LIN {X 0,Y 692.932,Z 1177.25,A -85,B 0,C 180,E1 3711.578,E2 3711.578} C_VEL
LIN {X 0,Y 695.46,Z 1123.55,A -85,B 0,C 180,E1 3717.284,E2 3717.284} C_VEL
LIN {X 0,Y 698.863,Z 1058.696,A -85,B 0,C 180,E1 3722.154,E2 3722.154} C_VEL
LIN {X 0,Y 702.382,Z 988.536,A -85,B 0,C 180,E1 3725.77,E2 3725.77} C_VEL
LIN {X 0,Y 705.082,Z 915.959,A -85,B 0,C 180,E1 3728.13,E2 3728.13} C_VEL
LIN {X 0,Y 704.438,Z 865.696,A -85,B 0,C 180,E1 3729.158,E2 3729.158} C_VEL
LIN {X 0,Y 689.914,Z 839.06,A -85,B 0,C 180,E1 3730.707,E2 3730.707} C_VEL
LIN {X 0,Y 690.212,Z 839.06,A -85,B 0,C 180,E1 3737.948,E2 3737.948} C_VEL
LIN {X 0,Y 690.254,Z 839.06,A -85,B 0,C 180,E1 3745.564,E2 3745.564} C_VEL
LIN {X 0,Y 690.297,Z 839.06,A -85,B 0,C 180,E1 3753.261,E2 3753.261} C_VEL
LIN {X 0,Y 690.399,Z 839.06,A -85,B 0,C 180,E1 3760.124,E2 3760.124} C_VEL
LIN {X 0,Y 690.82,Z 839.06,A -85,B 0,C 180,E1 3767.994,E2 3767.994} C_VEL
LIN {X 0,Y 690.331,Z 839.06,A -85,B 0,C 180,E1 3774.361,E2 3774.361} C_VEL
LIN {X 0,Y 690.785,Z 839.06,A -85,B 0,C 180,E1 3780.665,E2 3780.665} C_VEL
LIN {X 0,Y 690.621,Z 839.06,A -85,B 0,C 180,E1 3788.246,E2 3788.246} C_VEL
LIN {X 0,Y 690.564,Z 839.06,A -85,B 0,C 180,E1 3795.977,E2 3795.977} C_VEL
LIN {X 0,Y 690.789,Z 839.06,A -85,B 0,C 180,E1 3802.269,E2 3802.269} C_VEL
LIN {X 0,Y 682.311,Z 839.06,A -85,B 0,C 180,E1 3805.143,E2 3805.143} C_VEL
LIN {X 0,Y 682.215,Z 839.06,A -85,B 0,C 180,E1 3813.059,E2 3813.059} C_VEL
LIN {X 0,Y 682.25,Z 839.06,A -85,B 0,C 180,E1 3819.854,E2 3819.854} C_VEL
LIN {X 0,Y 682.232,Z 839.06,A -85,B 0,C 180,E1 3827.259,E2 3827.259} C_VEL
LIN {X 0,Y 682.2,Z 840.814,A -85,B 0,C 180,E1 3828.501,E2 3828.501} C_VEL
LIN {X 0,Y 699.805,Z 874.909,A -85,B 0,C 180,E1 3830.212,E2 3830.212} C_VEL
LIN {X 0,Y 698.506,Z 954.797,A -85,B 0,C 180,E1 3831.637,E2 3831.637} C_VEL
LIN {X 0,Y 695.396,Z 1024.983,A -85,B 0,C 180,E1 3834.062,E2 3834.062} C_VEL
LIN {X 0,Y 691.456,Z 1094.147,A -85,B 0,C 180,E1 3837.78,E2 3837.78} C_VEL
LIN {X 0,Y 687.671,Z 1156.924,A -85,B 0,C 180,E1 3842.648,E2 3842.648} C_VEL
LIN {X 0,Y 684.993,Z 1207.994,A -85,B 0,C 180,E1 3848.209,E2 3848.209} C_VEL
LIN {X 0,Y 683.695,Z 1243.057,A -85,B 0,C 180,E1 3853.555,E2 3853.555} C_VEL
LIN {X 0,Y 683.053,Z 1269.114,A -85,B 0,C 180,E1 3859.435,E2 3859.435} C_VEL
LIN {X 0,Y 683.019,Z 1282.874,A -85,B 0,C 180,E1 3864.9,E2 3864.9} C_VEL
LIN {X 0,Y 682.993,Z 1286.837,A -85,B 0,C 180,E1 3870.637,E2 3870.637} C_VEL
LIN {X 0,Y 683.016,Z 1280.509,A -85,B 0,C 180,E1 3876.381,E2 3876.381} C_VEL
LIN {X 0,Y 683.204,Z 1262.45,A -85,B 0,C 180,E1 3882.357,E2 3882.357} C_VEL
LIN {X 0,Y 684.024,Z 1233.434,A -85,B 0,C 180,E1 3888.103,E2 3888.103} C_VEL
LIN {X 0,Y 686.079,Z 1189.313,A -85,B 0,C 180,E1 3894.041,E2 3894.041} C_VEL
LIN {X 0,Y 689.325,Z 1131.43,A -85,B 0,C 180,E1 3899.539,E2 3899.539} C_VEL
LIN {X 0,Y 693.328,Z 1063.211,A -85,B 0,C 180,E1 3904.067,E2 3904.067} C_VEL
LIN {X 0,Y 697.084,Z 991.286,A -85,B 0,C 180,E1 3907.258,E2 3907.258} C_VEL
LIN {X 0,Y 699.503,Z 915.323,A -85,B 0,C 180,E1 3909.217,E2 3909.217} C_VEL
LIN {X 0,Y 698.507,Z 869.867,A -85,B 0,C 180,E1 3909.943,E2 3909.943} C_VEL
LIN {X 0,Y 682.019,Z 839.06,A -85,B 0,C 180,E1 3911.578,E2 3911.578} C_VEL
LIN {X 0,Y 682.178,Z 839.06,A -85,B 0,C 180,E1 3918.949,E2 3918.949} C_VEL
LIN {X 0,Y 682.569,Z 839.06,A -85,B 0,C 180,E1 3926.961,E2 3926.961} C_VEL
LIN {X 0,Y 682.913,Z 839.06,A -85,B 0,C 180,E1 3935.692,E2 3935.692} C_VEL
LIN {X 0,Y 682.634,Z 839.06,A -85,B 0,C 180,E1 3945.332,E2 3945.332} C_VEL
LIN {X 0,Y 682.779,Z 839.06,A -85,B 0,C 180,E1 3952.943,E2 3952.943} C_VEL
LIN {X 0,Y 682.878,Z 839.06,A -85,B 0,C 180,E1 3960.6,E2 3960.6} C_VEL
LIN {X 0,Y 682.689,Z 839.06,A -85,B 0,C 180,E1 3968.283,E2 3968.283} C_VEL
LIN {X 0,Y 682.549,Z 839.06,A -85,B 0,C 180,E1 3976.094,E2 3976.094} C_VEL
LIN {X 0,Y 682.553,Z 839.06,A -85,B 0,C 180,E1 3984.241,E2 3984.241} C_VEL
LIN {X 0,Y 682.499,Z 839.06,A -85,B 0,C 180,E1 3991.451,E2 3991.451} C_VEL
LIN {X 0,Y 682.274,Z 839.06,A -85,B 0,C 180,E1 3999.856,E2 3999.856} C_VEL
LIN {X 0,Y 682.267,Z 839.06,A -85,B 0,C 180,E1 4007.261,E2 4007.261} C_VEL
LIN {X 0,Y 682.009,Z 840.075,A -85,B 0,C 180,E1 4008.844,E2 4008.844} C_VEL
LIN {X 0,Y 699.791,Z 875.302,A -85,B 0,C 180,E1 4010.587,E2 4010.587} C_VEL
LIN {X 0,Y 697.423,Z 949.803,A -85,B 0,C 180,E1 4012.314,E2 4012.314} C_VEL
LIN {X 0,Y 693.842,Z 1023.138,A -85,B 0,C 180,E1 4015.353,E2 4015.353} C_VEL
LIN {X 0,Y 689.742,Z 1092.093,A -85,B 0,C 180,E1 4019.695,E2 4019.695} C_VEL
LIN {X 0,Y 686.311,Z 1151.955,A -85,B 0,C 180,E1 4025.098,E2 4025.098} C_VEL
LIN {X 0,Y 684.292,Z 1196.409,A -85,B 0,C 180,E1 4030.752,E2 4030.752} C_VEL
LIN {X 0,Y 683.279,Z 1227.921,A -85,B 0,C 180,E1 4036.509,E2 4036.509} C_VEL
LIN {X 0,Y 683.044,Z 1247.743,A -85,B 0,C 180,E1 4042.336,E2 4042.336} C_VEL
LIN {X 0,Y 682.885,Z 1256.414,A -85,B 0,C 180,E1 4048.089,E2 4048.089} C_VEL
LIN {X 0,Y 683.305,Z 1255.315,A -85,B 0,C 180,E1 4053.184,E2 4053.184} C_VEL
LIN {X 0,Y 683.118,Z 1242.086,A -85,B 0,C 180,E1 4059.594,E2 4059.594} C_VEL
LIN {X 0,Y 683.635,Z 1217.038,A -85,B 0,C 180,E1 4065.656,E2 4065.656} C_VEL
LIN {X 0,Y 685.159,Z 1177.253,A -85,B 0,C 180,E1 4071.835,E2 4071.835} C_VEL
LIN {X 0,Y 687.981,Z 1123.935,A -85,B 0,C 180,E1 4077.571,E2 4077.571} C_VEL
LIN {X 0,Y 691.853,Z 1058.702,A -85,B 0,C 180,E1 4082.52,E2 4082.52} C_VEL
LIN {X 0,Y 695.752,Z 988.547,A -85,B 0,C 180,E1 4086.164,E2 4086.164} C_VEL
LIN {X 0,Y 698.787,Z 915.966,A -85,B 0,C 180,E1 4088.536,E2 4088.536} C_VEL
LIN {X 0,Y 698.258,Z 869.263,A -85,B 0,C 180,E1 4089.52,E2 4089.52} C_VEL
LIN {X 0,Y 681.933,Z 839.06,A -85,B 0,C 180,E1 4091.286,E2 4091.286} C_VEL
LIN {X 0,Y 682.188,Z 839.06,A -85,B 0,C 180,E1 4098.201,E2 4098.201} C_VEL
LIN {X 0,Y 682.26,Z 839.06,A -85,B 0,C 180,E1 4105.499,E2 4105.499} C_VEL
LIN {X 0,Y 682.382,Z 839.06,A -85,B 0,C 180,E1 4112.925,E2 4112.925} C_VEL
LIN {X 0,Y 682.454,Z 839.06,A -85,B 0,C 180,E1 4119.882,E2 4119.882} C_VEL
LIN {X 0,Y 682.856,Z 839.06,A -85,B 0,C 180,E1 4127.852,E2 4127.852} C_VEL
LIN {X 0,Y 682.342,Z 839.06,A -85,B 0,C 180,E1 4134.294,E2 4134.294} C_VEL
LIN {X 0,Y 682.778,Z 839.06,A -85,B 0,C 180,E1 4140.673,E2 4140.673} C_VEL
LIN {X 0,Y 682.577,Z 839.06,A -85,B 0,C 180,E1 4148.344,E2 4148.344} C_VEL
LIN {X 0,Y 682.502,Z 839.06,A -85,B 0,C 180,E1 4156.171,E2 4156.171} C_VEL
LIN {X 0,Y 682.467,Z 839.06,A -85,B 0,C 180,E1 4164.325,E2 4164.325} C_VEL
LIN {X 0,Y 682.311,Z 839.06,A -85,B 0,C 180,E1 4165.143,E2 4165.143} C_VEL
LIN {X 0,Y 674.452,Z 839.06,A -85,B 0,C 180,E1 4168.067,E2 4168.067} C_VEL
LIN {X 0,Y 674.515,Z 839.06,A -85,B 0,C 180,E1 4176.967,E2 4176.967} C_VEL
LIN {X 0,Y 674.602,Z 839.06,A -85,B 0,C 180,E1 4185.16,E2 4185.16} C_VEL
LIN {X 0,Y 674.305,Z 840.847,A -85,B 0,C 180,E1 4187.906,E2 4187.906} C_VEL
LIN {X 0,Y 693.642,Z 877.2,A -85,B 0,C 180,E1 4189.817,E2 4189.817} C_VEL
LIN {X 0,Y 692.099,Z 956.399,A -85,B 0,C 180,E1 4191.263,E2 4191.263} C_VEL
LIN {X 0,Y 688.682,Z 1026.317,A -85,B 0,C 180,E1 4193.718,E2 4193.718} C_VEL
LIN {X 0,Y 684.318,Z 1095.736,A -85,B 0,C 180,E1 4197.511,E2 4197.511} C_VEL
LIN {X 0,Y 680.11,Z 1159.026,A -85,B 0,C 180,E1 4202.515,E2 4202.515} C_VEL
LIN {X 0,Y 677.106,Z 1210.63,A -85,B 0,C 180,E1 4208.288,E2 4208.288} C_VEL
LIN {X 0,Y 675.555,Z 1246.593,A -85,B 0,C 180,E1 4214.021,E2 4214.021} C_VEL
LIN {X 0,Y 675.033,Z 1270.262,A -85,B 0,C 180,E1 4219.636,E2 4219.636} C_VEL
LIN {X 0,Y 674.821,Z 1283.82,A -85,B 0,C 180,E1 4225.484,E2 4225.484} C_VEL
LIN {X 0,Y 675.007,Z 1286.837,A -85,B 0,C 180,E1 4230.645,E2 4230.645} C_VEL
LIN {X 0,Y 675.009,Z 1280.509,A -85,B 0,C 180,E1 4236.457,E2 4236.457} C_VEL
LIN {X 0,Y 675.267,Z 1263.15,A -85,B 0,C 180,E1 4242.332,E2 4242.332} C_VEL
LIN {X 0,Y 676.091,Z 1233.436,A -85,B 0,C 180,E1 4248.323,E2 4248.323} C_VEL
LIN {X 0,Y 678.369,Z 1190.121,A -85,B 0,C 180,E1 4254.236,E2 4254.236} C_VEL
LIN {X 0,Y 681.89,Z 1133.351,A -85,B 0,C 180,E1 4259.727,E2 4259.727} C_VEL
LIN {X 0,Y 686.284,Z 1066.871,A -85,B 0,C 180,E1 4264.252,E2 4264.252} C_VEL
LIN {X 0,Y 690.378,Z 995.277,A -85,B 0,C 180,E1 4267.523,E2 4267.523} C_VEL
LIN {X 0,Y 693.157,Z 919.424,A -85,B 0,C 180,E1 4269.565,E2 4269.565} C_VEL
LIN {X 0,Y 692.205,Z 872.842,A -85,B 0,C 180,E1 4270.342,E2 4270.342} C_VEL
LIN {X 0,Y 674.122,Z 839.06,A -85,B 0,C 180,E1 4272.34,E2 4272.34} C_VEL
LIN {X 0,Y 674.296,Z 839.06,A -85,B 0,C 180,E1 4280.066,E2 4280.066} C_VEL
LIN {X 0,Y 674.685,Z 839.06,A -85,B 0,C 180,E1 4288.055,E2 4288.055} C_VEL
LIN {X 0,Y 674.926,Z 839.06,A -85,B 0,C 180,E1 4295.641,E2 4295.641} C_VEL
LIN {X 0,Y 674.691,Z 839.06,A -85,B 0,C 180,E1 4304.975,E2 4304.975} C_VEL
LIN {X 0,Y 674.795,Z 839.06,A -85,B 0,C 180,E1 4312.859,E2 4312.859} C_VEL
LIN {X 0,Y 674.89,Z 839.06,A -85,B 0,C 180,E1 4320.607,E2 4320.607} C_VEL
LIN {X 0,Y 674.68,Z 839.06,A -85,B 0,C 180,E1 4328.368,E2 4328.368} C_VEL
LIN {X 0,Y 674.464,Z 839.06,A -85,B 0,C 180,E1 4336.292,E2 4336.292} C_VEL
LIN {X 0,Y 674.476,Z 839.06,A -85,B 0,C 180,E1 4344.551,E2 4344.551} C_VEL
LIN {X 0,Y 674.288,Z 839.06,A -85,B 0,C 180,E1 4352.403,E2 4352.403} C_VEL
LIN {X 0,Y 674.293,Z 839.06,A -85,B 0,C 180,E1 4359.838,E2 4359.838} C_VEL
LIN {X 0,Y 674.344,Z 839.06,A -85,B 0,C 180,E1 4366.934,E2 4366.934} C_VEL
LIN {X 0,Y 674.31,Z 841.198,A -85,B 0,C 180,E1 4368.286,E2 4368.286} C_VEL
LIN {X 0,Y 693.579,Z 878.428,A -85,B 0,C 180,E1 4370.214,E2 4370.214} C_VEL
LIN {X 0,Y 690.91,Z 951.54,A -85,B 0,C 180,E1 4371.958,E2 4371.958} C_VEL
LIN {X 0,Y 686.923,Z 1025.135,A -85,B 0,C 180,E1 4375.067,E2 4375.067} C_VEL
LIN {X 0,Y 682.415,Z 1093.761,A -85,B 0,C 180,E1 4379.469,E2 4379.469} C_VEL
LIN {X 0,Y 678.68,Z 1152.869,A -85,B 0,C 180,E1 4384.9,E2 4384.9} C_VEL
LIN {X 0,Y 676.445,Z 1196.769,A -85,B 0,C 180,E1 4390.576,E2 4390.576} C_VEL
LIN {X 0,Y 675.373,Z 1227.92,A -85,B 0,C 180,E1 4396.348,E2 4396.348} C_VEL
LIN {X 0,Y 675.088,Z 1247.739,A -85,B 0,C 180,E1 4402.245,E2 4402.245} C_VEL
LIN {X 0,Y 674.893,Z 1256.413,A -85,B 0,C 180,E1 4408.066,E2 4408.066} C_VEL
LIN {X 0,Y 675.307,Z 1255.315,A -85,B 0,C 180,E1 4413.221,E2 4413.221} C_VEL
LIN {X 0,Y 675.088,Z 1242.089,A -85,B 0,C 180,E1 4419.709,E2 4419.709} C_VEL
LIN {X 0,Y 675.703,Z 1217.838,A -85,B 0,C 180,E1 4425.691,E2 4425.691} C_VEL
LIN {X 0,Y 677.352,Z 1179.112,A -85,B 0,C 180,E1 4431.859,E2 4431.859} C_VEL
LIN {X 0,Y 680.405,Z 1126.459,A -85,B 0,C 180,E1 4437.668,E2 4437.668} C_VEL
LIN {X 0,Y 684.549,Z 1062.394,A -85,B 0,C 180,E1 4442.66,E2 4442.66} C_VEL
LIN {X 0,Y 688.958,Z 991.893,A -85,B 0,C 180,E1 4446.425,E2 4446.425} C_VEL
LIN {X 0,Y 692.432,Z 917.33,A -85,B 0,C 180,E1 4448.922,E2 4448.922} C_VEL
LIN {X 0,Y 692.118,Z 872.536,A -85,B 0,C 180,E1 4449.889,E2 4449.889} C_VEL
LIN {X 0,Y 674.035,Z 839.06,A -85,B 0,C 180,E1 4451.839,E2 4451.839} C_VEL
LIN {X 0,Y 674.187,Z 839.06,A -85,B 0,C 180,E1 4458.968,E2 4458.968} C_VEL
LIN {X 0,Y 674.214,Z 839.06,A -85,B 0,C 180,E1 4466.586,E2 4466.586} C_VEL
LIN {X 0,Y 674.299,Z 839.06,A -85,B 0,C 180,E1 4474.017,E2 4474.017} C_VEL
LIN {X 0,Y 674.246,Z 839.06,A -85,B 0,C 180,E1 4480.996,E2 4480.996} C_VEL
LIN {X 0,Y 674.848,Z 839.06,A -85,B 0,C 180,E1 4488.113,E2 4488.113} C_VEL
LIN {X 0,Y 674.372,Z 839.06,A -85,B 0,C 180,E1 4494.227,E2 4494.227} C_VEL
LIN {X 0,Y 674.789,Z 839.06,A -85,B 0,C 180,E1 4500.681,E2 4500.681} C_VEL
LIN {X 0,Y 674.534,Z 839.06,A -85,B 0,C 180,E1 4508.444,E2 4508.444} C_VEL
LIN {X 0,Y 674.419,Z 839.06,A -85,B 0,C 180,E1 4516.371,E2 4516.371} C_VEL
LIN {X 0,Y 674.398,Z 839.06,A -85,B 0,C 180,E1 4524.635,E2 4524.635} C_VEL
LIN {X 0,Y 674.452,Z 839.06,A -85,B 0,C 180,E1 4528.067,E2 4528.067} C_VEL
LIN {X 0,Y 666.458,Z 839.06,A -85,B 0,C 180,E1 4531.02,E2 4531.02} C_VEL
LIN {X 0,Y 666.377,Z 839.06,A -85,B 0,C 180,E1 4538.812,E2 4538.812} C_VEL
LIN {X 0,Y 666.232,Z 839.091,A -85,B 0,C 180,E1 4547.25,E2 4547.25} C_VEL
LIN {X 0,Y 687.479,Z 881.775,A -85,B 0,C 180,E1 4549.444,E2 4549.444} C_VEL
LIN {X 0,Y 685.68,Z 959.359,A -85,B 0,C 180,E1 4550.923,E2 4550.923} C_VEL
LIN {X 0,Y 681.852,Z 1030.289,A -85,B 0,C 180,E1 4553.484,E2 4553.484} C_VEL
LIN {X 0,Y 677.008,Z 1099.887,A -85,B 0,C 180,E1 4557.404,E2 4557.404} C_VEL
LIN {X 0,Y 672.432,Z 1162.703,A -85,B 0,C 180,E1 4562.545,E2 4562.545} C_VEL
LIN {X 0,Y 669.231,Z 1212.573,A -85,B 0,C 180,E1 4568.297,E2 4568.297} C_VEL
LIN {X 0,Y 667.692,Z 1246.594,A -85,B 0,C 180,E1 4573.828,E2 4573.828} C_VEL
LIN {X 0,Y 667.095,Z 1270.261,A -85,B 0,C 180,E1 4579.511,E2 4579.511} C_VEL
LIN {X 0,Y 666.836,Z 1283.817,A -85,B 0,C 180,E1 4585.43,E2 4585.43} C_VEL
LIN {X 0,Y 667.002,Z 1286.837,A -85,B 0,C 180,E1 4590.652,E2 4590.652} C_VEL
LIN {X 0,Y 666.991,Z 1280.509,A -85,B 0,C 180,E1 4596.535,E2 4596.535} C_VEL
LIN {X 0,Y 667.252,Z 1263.15,A -85,B 0,C 180,E1 4602.483,E2 4602.483} C_VEL
LIN {X 0,Y 668.2,Z 1233.438,A -85,B 0,C 180,E1 4608.547,E2 4608.547} C_VEL
LIN {X 0,Y 670.646,Z 1191.149,A -85,B 0,C 180,E1 4614.41,E2 4614.41} C_VEL
LIN {X 0,Y 674.466,Z 1135.205,A -85,B 0,C 180,E1 4619.924,E2 4619.924} C_VEL
LIN {X 0,Y 679.222,Z 1069.408,A -85,B 0,C 180,E1 4624.499,E2 4624.499} C_VEL
LIN {X 0,Y 683.764,Z 997.734,A -85,B 0,C 180,E1 4627.848,E2 4627.848} C_VEL
LIN {X 0,Y 686.867,Z 921.844,A -85,B 0,C 180,E1 4629.948,E2 4629.948} C_VEL
LIN {X 0,Y 686.237,Z 876.309,A -85,B 0,C 180,E1 4630.719,E2 4630.719} C_VEL
LIN {X 0,Y 666.244,Z 839.06,A -85,B 0,C 180,E1 4632.798,E2 4632.798} C_VEL
LIN {X 0,Y 666.548,Z 839.06,A -85,B 0,C 180,E1 4641.792,E2 4641.792} C_VEL
LIN {X 0,Y 666.757,Z 839.06,A -85,B 0,C 180,E1 4650.667,E2 4650.667} C_VEL
LIN {X 0,Y 666.275,Z 839.06,A -85,B 0,C 180,E1 4657.89,E2 4657.89} C_VEL
LIN {X 0,Y 666.378,Z 839.06,A -85,B 0,C 180,E1 4666.13,E2 4666.13} C_VEL
LIN {X 0,Y 666.811,Z 839.06,A -85,B 0,C 180,E1 4672.773,E2 4672.773} C_VEL
LIN {X 0,Y 666.88,Z 839.06,A -85,B 0,C 180,E1 4680.614,E2 4680.614} C_VEL
LIN {X 0,Y 666.66,Z 839.06,A -85,B 0,C 180,E1 4688.469,E2 4688.469} C_VEL
LIN {X 0,Y 666.387,Z 839.06,A -85,B 0,C 180,E1 4696.495,E2 4696.495} C_VEL
LIN {X 0,Y 666.402,Z 839.06,A -85,B 0,C 180,E1 4704.868,E2 4704.868} C_VEL
LIN {X 0,Y 666.314,Z 839.06,A -85,B 0,C 180,E1 4712.306,E2 4712.306} C_VEL
LIN {X 0,Y 666.216,Z 839.06,A -85,B 0,C 180,E1 4720.42,E2 4720.42} C_VEL
LIN {X 0,Y 666.372,Z 840.921,A -85,B 0,C 180,E1 4727.672,E2 4727.672} C_VEL
LIN {X 0,Y 687.346,Z 882.175,A -85,B 0,C 180,E1 4729.845,E2 4729.845} C_VEL
LIN {X 0,Y 684.359,Z 955.318,A -85,B 0,C 180,E1 4731.666,E2 4731.666} C_VEL
LIN {X 0,Y 680.02,Z 1027.293,A -85,B 0,C 180,E1 4734.784,E2 4734.784} C_VEL
LIN {X 0,Y 675.154,Z 1094.568,A -85,B 0,C 180,E1 4739.172,E2 4739.172} C_VEL
LIN {X 0,Y 671.086,Z 1152.861,A -85,B 0,C 180,E1 4744.596,E2 4744.596} C_VEL
LIN {X 0,Y 668.576,Z 1197.702,A -85,B 0,C 180,E1 4750.484,E2 4750.484} C_VEL
LIN {X 0,Y 667.35,Z 1229.276,A -85,B 0,C 180,E1 4756.516,E2 4756.516} C_VEL
LIN {X 0,Y 667.148,Z 1247.735,A -85,B 0,C 180,E1 4762.152,E2 4762.152} C_VEL
LIN {X 0,Y 666.898,Z 1256.413,A -85,B 0,C 180,E1 4768.043,E2 4768.043} C_VEL
LIN {X 0,Y 667.282,Z 1255.316,A -85,B 0,C 180,E1 4773.26,E2 4773.26} C_VEL
LIN {X 0,Y 667.071,Z 1242.091,A -85,B 0,C 180,E1 4779.827,E2 4779.827} C_VEL
LIN {X 0,Y 667.731,Z 1218.101,A -85,B 0,C 180,E1 4785.832,E2 4785.832} C_VEL
LIN {X 0,Y 669.579,Z 1178.979,A -85,B 0,C 180,E1 4792.143,E2 4792.143} C_VEL
LIN {X 0,Y 672.944,Z 1127.047,A -85,B 0,C 180,E1 4797.946,E2 4797.946} C_VEL
LIN {X 0,Y 677.458,Z 1063.829,A -85,B 0,C 180,E1 4802.946,E2 4802.946} C_VEL
LIN {X 0,Y 682.302,Z 993.163,A -85,B 0,C 180,E1 4806.78,E2 4806.78} C_VEL
LIN {X 0,Y 686.135,Z 918.435,A -85,B 0,C 180,E1 4809.319,E2 4809.319} C_VEL
LIN {X 0,Y 685.993,Z 875.954,A -85,B 0,C 180,E1 4810.263,E2 4810.263} C_VEL
LIN {X 0,Y 666.16,Z 839.06,A -85,B 0,C 180,E1 4812.308,E2 4812.308} C_VEL
LIN {X 0,Y 666.264,Z 839.06,A -85,B 0,C 180,E1 4819.757,E2 4819.757} C_VEL
LIN {X 0,Y 666.324,Z 839.06,A -85,B 0,C 180,E1 4827.695,E2 4827.695} C_VEL
LIN {X 0,Y 666.377,Z 839.06,A -85,B 0,C 180,E1 4835.131,E2 4835.131} C_VEL
LIN {X 0,Y 666.559,Z 839.06,A -85,B 0,C 180,E1 4843.509,E2 4843.509} C_VEL
LIN {X 0,Y 667.15,Z 839.06,A -85,B 0,C 180,E1 4851.829,E2 4851.829} C_VEL
LIN {X 0,Y 666.782,Z 839.06,A -85,B 0,C 180,E1 4860.689,E2 4860.689} C_VEL
LIN {X 0,Y 666.514,Z 839.06,A -85,B 0,C 180,E1 4868.547,E2 4868.547} C_VEL
LIN {X 0,Y 666.357,Z 839.06,A -85,B 0,C 180,E1 4876.574,E2 4876.574} C_VEL
LIN {X 0,Y 666.334,Z 839.06,A -85,B 0,C 180,E1 4884.954,E2 4884.954} C_VEL
LIN {X 0,Y 666.458,Z 839.06,A -85,B 0,C 180,E1 4891.02,E2 4891.02} C_VEL
LIN {X 0,Y 658.161,Z 839.06,A -85,B 0,C 180,E1 4894.011,E2 4894.011} C_VEL
LIN {X 0,Y 658.119,Z 839.06,A -85,B 0,C 180,E1 4901.437,E2 4901.437} C_VEL
LIN {X 0,Y 658.519,Z 840.38,A -85,B 0,C 180,E1 4906.646,E2 4906.646} C_VEL
LIN {X 0,Y 681.369,Z 885.346,A -85,B 0,C 180,E1 4909.051,E2 4909.051} C_VEL
LIN {X 0,Y 679.23,Z 963.177,A -85,B 0,C 180,E1 4910.6,E2 4910.6} C_VEL
LIN {X 0,Y 674.995,Z 1033.456,A -85,B 0,C 180,E1 4913.219,E2 4913.219} C_VEL
LIN {X 0,Y 669.773,Z 1102.545,A -85,B 0,C 180,E1 4917.21,E2 4917.21} C_VEL
LIN {X 0,Y 664.788,Z 1165.331,A -85,B 0,C 180,E1 4922.476,E2 4922.476} C_VEL
LIN {X 0,Y 661.433,Z 1213.351,A -85,B 0,C 180,E1 4928.141,E2 4928.141} C_VEL
LIN {X 0,Y 659.682,Z 1248.333,A -85,B 0,C 180,E1 4933.97,E2 4933.97} C_VEL
LIN {X 0,Y 659.134,Z 1270.261,A -85,B 0,C 180,E1 4939.383,E2 4939.383} C_VEL
LIN {X 0,Y 658.852,Z 1283.814,A -85,B 0,C 180,E1 4945.375,E2 4945.375} C_VEL
LIN {X 0,Y 659.005,Z 1286.837,A -85,B 0,C 180,E1 4950.66,E2 4950.66} C_VEL
LIN {X 0,Y 658.982,Z 1280.509,A -85,B 0,C 180,E1 4956.615,E2 4956.615} C_VEL
LIN {X 0,Y 659.274,Z 1263.149,A -85,B 0,C 180,E1 4962.636,E2 4962.636} C_VEL
LIN {X 0,Y 660.338,Z 1233.439,A -85,B 0,C 180,E1 4968.776,E2 4968.776} C_VEL
LIN {X 0,Y 662.963,Z 1191.22,A -85,B 0,C 180,E1 4974.703,E2 4974.703} C_VEL
LIN {X 0,Y 667.23,Z 1135.204,A -85,B 0,C 180,E1 4980.282,E2 4980.282} C_VEL
LIN {X 0,Y 672.382,Z 1069.327,A -85,B 0,C 180,E1 4984.905,E2 4984.905} C_VEL
LIN {X 0,Y 677.281,Z 998.842,A -85,B 0,C 180,E1 4988.229,E2 4988.229} C_VEL
LIN {X 0,Y 680.674,Z 923.249,A -85,B 0,C 180,E1 4990.356,E2 4990.356} C_VEL
LIN {X 0,Y 680.091,Z 879.557,A -85,B 0,C 180,E1 4991.122,E2 4991.122} C_VEL
LIN {X 0,Y 658.392,Z 839.06,A -85,B 0,C 180,E1 4993.403,E2 4993.403} C_VEL
LIN {X 0,Y 658.593,Z 839.06,A -85,B 0,C 180,E1 5002.68,E2 5002.68} C_VEL
LIN {X 0,Y 658.714,Z 839.06,A -85,B 0,C 180,E1 5010.273,E2 5010.273} C_VEL
LIN {X 0,Y 658.349,Z 839.06,A -85,B 0,C 180,E1 5017.61,E2 5017.61} C_VEL
LIN {X 0,Y 658.419,Z 839.06,A -85,B 0,C 180,E1 5025.959,E2 5025.959} C_VEL
LIN {X 0,Y 658.84,Z 839.06,A -85,B 0,C 180,E1 5032.685,E2 5032.685} C_VEL
LIN {X 0,Y 658.893,Z 839.06,A -85,B 0,C 180,E1 5040.622,E2 5040.622} C_VEL
LIN {X 0,Y 658.615,Z 839.06,A -85,B 0,C 180,E1 5048.573,E2 5048.573} C_VEL
LIN {X 0,Y 658.322,Z 839.06,A -85,B 0,C 180,E1 5056.703,E2 5056.703} C_VEL
LIN {X 0,Y 658.355,Z 839.06,A -85,B 0,C 180,E1 5065.193,E2 5065.193} C_VEL
LIN {X 0,Y 658.239,Z 839.06,A -85,B 0,C 180,E1 5072.751,E2 5072.751} C_VEL
LIN {X 0,Y 658.283,Z 839.06,A -85,B 0,C 180,E1 5079.414,E2 5079.414} C_VEL
LIN {X 0,Y 658.406,Z 840.317,A -85,B 0,C 180,E1 5087.03,E2 5087.03} C_VEL
LIN {X 0,Y 681.168,Z 883.875,A -85,B 0,C 180,E1 5089.438,E2 5089.438} C_VEL
LIN {X 0,Y 677.962,Z 955.757,A -85,B 0,C 180,E1 5091.254,E2 5091.254} C_VEL
LIN {X 0,Y 673.28,Z 1027.237,A -85,B 0,C 180,E1 5094.376,E2 5094.376} C_VEL
LIN {X 0,Y 667.956,Z 1095.139,A -85,B 0,C 180,E1 5098.85,E2 5098.85} C_VEL
LIN {X 0,Y 663.501,Z 1153.556,A -85,B 0,C 180,E1 5104.364,E2 5104.364} C_VEL
LIN {X 0,Y 660.807,Z 1197.697,A -85,B 0,C 180,E1 5110.245,E2 5110.245} C_VEL
LIN {X 0,Y 659.438,Z 1229.274,A -85,B 0,C 180,E1 5116.351,E2 5116.351} C_VEL
LIN {X 0,Y 658.918,Z 1249.247,A -85,B 0,C 180,E1 5122.72,E2 5122.72} C_VEL
LIN {X 0,Y 658.934,Z 1256.413,A -85,B 0,C 180,E1 5128.019,E2 5128.019} C_VEL
LIN {X 0,Y 659.272,Z 1255.316,A -85,B 0,C 180,E1 5133.3,E2 5133.3} C_VEL
LIN {X 0,Y 659.206,Z 1243.515,A -85,B 0,C 180,E1 5139.456,E2 5139.456} C_VEL
LIN {X 0,Y 659.861,Z 1219.827,A -85,B 0,C 180,E1 5145.683,E2 5145.683} C_VEL
LIN {X 0,Y 661.723,Z 1181.976,A -85,B 0,C 180,E1 5152.003,E2 5152.003} C_VEL
LIN {X 0,Y 665.354,Z 1130.1,A -85,B 0,C 180,E1 5157.999,E2 5157.999} C_VEL
LIN {X 0,Y 670.289,Z 1066.54,A -85,B 0,C 180,E1 5163.155,E2 5163.155} C_VEL
LIN {X 0,Y 675.571,Z 996.448,A -85,B 0,C 180,E1 5167.052,E2 5167.052} C_VEL
LIN {X 0,Y 679.684,Z 922.282,A -85,B 0,C 180,E1 5169.66,E2 5169.66} C_VEL
LIN {X 0,Y 679.893,Z 879.418,A -85,B 0,C 180,E1 5170.644,E2 5170.644} C_VEL
LIN {X 0,Y 658.197,Z 839.06,A -85,B 0,C 180,E1 5172.921,E2 5172.921} C_VEL
LIN {X 0,Y 658.322,Z 839.06,A -85,B 0,C 180,E1 5180.72,E2 5180.72} C_VEL
LIN {X 0,Y 658.547,Z 839.06,A -85,B 0,C 180,E1 5189.822,E2 5189.822} C_VEL
LIN {X 0,Y 658.536,Z 839.06,A -85,B 0,C 180,E1 5199.118,E2 5199.118} C_VEL
LIN {X 0,Y 658.866,Z 839.06,A -85,B 0,C 180,E1 5207.403,E2 5207.403} C_VEL
LIN {X 0,Y 658.425,Z 839.06,A -85,B 0,C 180,E1 5214.086,E2 5214.086} C_VEL
LIN {X 0,Y 658.782,Z 839.06,A -85,B 0,C 180,E1 5220.698,E2 5220.698} C_VEL
LIN {X 0,Y 658.472,Z 839.06,A -85,B 0,C 180,E1 5228.652,E2 5228.652} C_VEL
LIN {X 0,Y 658.281,Z 839.06,A -85,B 0,C 180,E1 5236.851,E2 5236.851} C_VEL
LIN {X 0,Y 658.399,Z 839.06,A -85,B 0,C 180,E1 5244.388,E2 5244.388} C_VEL
LIN {X 0,Y 658.215,Z 839.06,A -85,B 0,C 180,E1 5252.843,E2 5252.843} C_VEL
LIN {X 0,Y 658.161,Z 839.06,A -85,B 0,C 180,E1 5254.011,E2 5254.011} C_VEL
LIN {X 0,Y 650.34,Z 839.06,A -85,B 0,C 180,E1 5257.037,E2 5257.037} C_VEL
LIN {X 0,Y 650.503,Z 840.565,A -85,B 0,C 180,E1 5265.978,E2 5265.978} C_VEL
LIN {X 0,Y 675.297,Z 888.284,A -85,B 0,C 180,E1 5268.643,E2 5268.643} C_VEL
LIN {X 0,Y 672.823,Z 966.353,A -85,B 0,C 180,E1 5270.252,E2 5270.252} C_VEL
LIN {X 0,Y 668.035,Z 1038.706,A -85,B 0,C 180,E1 5273.053,E2 5273.053} C_VEL
LIN {X 0,Y 662.214,Z 1108.806,A -85,B 0,C 180,E1 5277.272,E2 5277.272} C_VEL
LIN {X 0,Y 656.953,Z 1170.73,A -85,B 0,C 180,E1 5282.692,E2 5282.692} C_VEL
LIN {X 0,Y 653.299,Z 1219.103,A -85,B 0,C 180,E1 5288.702,E2 5288.702} C_VEL
LIN {X 0,Y 651.611,Z 1251.592,A -85,B 0,C 180,E1 5294.46,E2 5294.46} C_VEL
LIN {X 0,Y 650.988,Z 1272.224,A -85,B 0,C 180,E1 5299.927,E2 5299.927} C_VEL
LIN {X 0,Y 650.869,Z 1283.811,A -85,B 0,C 180,E1 5305.318,E2 5305.318} C_VEL
LIN {X 0,Y 650.999,Z 1286.837,A -85,B 0,C 180,E1 5310.668,E2 5310.668} C_VEL
LIN {X 0,Y 650.989,Z 1280.509,A -85,B 0,C 180,E1 5316.696,E2 5316.696} C_VEL
LIN {X 0,Y 651.274,Z 1263.148,A -85,B 0,C 180,E1 5322.794,E2 5322.794} C_VEL
LIN {X 0,Y 652.485,Z 1233.807,A -85,B 0,C 180,E1 5328.945,E2 5328.945} C_VEL
LIN {X 0,Y 655.363,Z 1191.222,A -85,B 0,C 180,E1 5335.009,E2 5335.009} C_VEL
LIN {X 0,Y 659.971,Z 1135.096,A -85,B 0,C 180,E1 5340.66,E2 5340.66} C_VEL
LIN {X 0,Y 665.706,Z 1068.504,A -85,B 0,C 180,E1 5345.36,E2 5345.36} C_VEL
LIN {X 0,Y 670.953,Z 997.699,A -85,B 0,C 180,E1 5348.704,E2 5348.704} C_VEL
LIN {X 0,Y 674.615,Z 922.239,A -85,B 0,C 180,E1 5350.816,E2 5350.816} C_VEL
LIN {X 0,Y 674.108,Z 882.848,A -85,B 0,C 180,E1 5351.521,E2 5351.521} C_VEL
LIN {X 0,Y 650.371,Z 839.06,A -85,B 0,C 180,E1 5354.127,E2 5354.127} C_VEL
LIN {X 0,Y 650.567,Z 839.06,A -85,B 0,C 180,E1 5363.618,E2 5363.618} C_VEL
LIN {X 0,Y 650.634,Z 839.06,A -85,B 0,C 180,E1 5371.399,E2 5371.399} C_VEL
LIN {X 0,Y 650.103,Z 839.06,A -85,B 0,C 180,E1 5378.752,E2 5378.752} C_VEL
LIN {X 0,Y 650.433,Z 839.06,A -85,B 0,C 180,E1 5385.783,E2 5385.783} C_VEL
LIN {X 0,Y 650.864,Z 839.06,A -85,B 0,C 180,E1 5392.595,E2 5392.595} C_VEL
LIN {X 0,Y 650.884,Z 839.06,A -85,B 0,C 180,E1 5400.629,E2 5400.629} C_VEL
LIN {X 0,Y 650.572,Z 839.06,A -85,B 0,C 180,E1 5408.68,E2 5408.68} C_VEL
LIN {X 0,Y 650.279,Z 839.06,A -85,B 0,C 180,E1 5416.916,E2 5416.916} C_VEL
LIN {X 0,Y 650.509,Z 839.06,A -85,B 0,C 180,E1 5424.047,E2 5424.047} C_VEL
LIN {X 0,Y 650.381,Z 839.06,A -85,B 0,C 180,E1 5431.615,E2 5431.615} C_VEL
LIN {X 0,Y 650.197,Z 839.06,A -85,B 0,C 180,E1 5439.868,E2 5439.868} C_VEL
LIN {X 0,Y 650.478,Z 840.338,A -85,B 0,C 180,E1 5446.377,E2 5446.377} C_VEL
LIN {X 0,Y 674.998,Z 887.231,A -85,B 0,C 180,E1 5449.059,E2 5449.059} C_VEL
LIN {X 0,Y 671.445,Z 959.456,A -85,B 0,C 180,E1 5450.945,E2 5450.945} C_VEL
LIN {X 0,Y 666.306,Z 1030.452,A -85,B 0,C 180,E1 5454.136,E2 5454.136} C_VEL
LIN {X 0,Y 660.478,Z 1098.574,A -85,B 0,C 180,E1 5458.746,E2 5458.746} C_VEL
LIN {X 0,Y 655.703,Z 1156.843,A -85,B 0,C 180,E1 5464.418,E2 5464.418} C_VEL
LIN {X 0,Y 652.675,Z 1201.705,A -85,B 0,C 180,E1 5470.643,E2 5470.643} C_VEL
LIN {X 0,Y 651.374,Z 1230.63,A -85,B 0,C 180,E1 5476.522,E2 5476.522} C_VEL
LIN {X 0,Y 650.949,Z 1249.245,A -85,B 0,C 180,E1 5482.63,E2 5482.63} C_VEL
LIN {X 0,Y 650.939,Z 1256.413,A -85,B 0,C 180,E1 5487.995,E2 5487.995} C_VEL
LIN {X 0,Y 651.248,Z 1255.316,A -85,B 0,C 180,E1 5493.341,E2 5493.341} C_VEL
LIN {X 0,Y 651.265,Z 1244.036,A -85,B 0,C 180,E1 5499.391,E2 5499.391} C_VEL
LIN {X 0,Y 651.874,Z 1219.83,A -85,B 0,C 180,E1 5505.881,E2 5505.881} C_VEL
LIN {X 0,Y 653.975,Z 1181.98,A -85,B 0,C 180,E1 5512.278,E2 5512.278} C_VEL
LIN {X 0,Y 657.858,Z 1131.18,A -85,B 0,C 180,E1 5518.233,E2 5518.233} C_VEL
LIN {X 0,Y 663.239,Z 1067.899,A -85,B 0,C 180,E1 5523.457,E2 5523.457} C_VEL
LIN {X 0,Y 668.946,Z 998.017,A -85,B 0,C 180,E1 5527.407,E2 5527.407} C_VEL
LIN {X 0,Y 673.436,Z 923.376,A -85,B 0,C 180,E1 5530.071,E2 5530.071} C_VEL
LIN {X 0,Y 673.809,Z 882.793,A -85,B 0,C 180,E1 5531.03,E2 5531.03} C_VEL
LIN {X 0,Y 650.325,Z 839.06,A -85,B 0,C 180,E1 5533.569,E2 5533.569} C_VEL
LIN {X 0,Y 650.397,Z 839.06,A -85,B 0,C 180,E1 5541.866,E2 5541.866} C_VEL
LIN {X 0,Y 650.505,Z 839.06,A -85,B 0,C 180,E1 5551.063,E2 5551.063} C_VEL
LIN {X 0,Y 650.563,Z 839.06,A -85,B 0,C 180,E1 5558.85,E2 5558.85} C_VEL
LIN {X 0,Y 650.858,Z 839.06,A -85,B 0,C 180,E1 5567.245,E2 5567.245} C_VEL
LIN {X 0,Y 650.436,Z 839.06,A -85,B 0,C 180,E1 5574.013,E2 5574.013} C_VEL
LIN {X 0,Y 650.776,Z 839.06,A -85,B 0,C 180,E1 5580.706,E2 5580.706} C_VEL
LIN {X 0,Y 650.46,Z 839.06,A -85,B 0,C 180,E1 5588.759,E2 5588.759} C_VEL
LIN {X 0,Y 650.263,Z 839.06,A -85,B 0,C 180,E1 5596.997,E2 5596.997} C_VEL
LIN {X 0,Y 650.48,Z 839.06,A -85,B 0,C 180,E1 5604.132,E2 5604.132} C_VEL
LIN {X 0,Y 650.338,Z 839.06,A -85,B 0,C 180,E1 5611.707,E2 5611.707} C_VEL
LIN {X 0,Y 650.34,Z 839.06,A -85,B 0,C 180,E1 5617.037,E2 5617.037} C_VEL
LIN {X 0,Y 642.133,Z 839.06,A -85,B 0,C 180,E1 5620.107,E2 5620.107} C_VEL
LIN {X 0,Y 642.603,Z 840.862,A -85,B 0,C 180,E1 5625.298,E2 5625.298} C_VEL
LIN {X 0,Y 669.242,Z 891.705,A -85,B 0,C 180,E1 5628.234,E2 5628.234} C_VEL
LIN {X 0,Y 666.36,Z 970.383,A -85,B 0,C 180,E1 5629.922,E2 5629.922} C_VEL
LIN {X 0,Y 661.096,Z 1043.489,A -85,B 0,C 180,E1 5632.86,E2 5632.86} C_VEL
LIN {X 0,Y 654.916,Z 1112.348,A -85,B 0,C 180,E1 5637.139,E2 5637.139} C_VEL
LIN {X 0,Y 649.375,Z 1172.428,A -85,B 0,C 180,E1 5642.529,E2 5642.529} C_VEL
LIN {X 0,Y 645.468,Z 1220.365,A -85,B 0,C 180,E1 5648.62,E2 5648.62} C_VEL
LIN {X 0,Y 643.646,Z 1253.336,A -85,B 0,C 180,E1 5654.654,E2 5654.654} C_VEL
LIN {X 0,Y 642.977,Z 1274.164,A -85,B 0,C 180,E1 5660.487,E2 5660.487} C_VEL
LIN {X 0,Y 642.902,Z 1283.808,A -85,B 0,C 180,E1 5665.26,E2 5665.26} C_VEL
LIN {X 0,Y 643.018,Z 1286.837,A -85,B 0,C 180,E1 5670.677,E2 5670.677} C_VEL
LIN {X 0,Y 642.997,Z 1280.535,A -85,B 0,C 180,E1 5676.767,E2 5676.767} C_VEL
LIN {X 0,Y 643.294,Z 1263.147,A -85,B 0,C 180,E1 5682.956,E2 5682.956} C_VEL
LIN {X 0,Y 644.541,Z 1235.754,A -85,B 0,C 180,E1 5688.838,E2 5688.838} C_VEL
LIN {X 0,Y 647.602,Z 1193.328,A -85,B 0,C 180,E1 5695.065,E2 5695.065} C_VEL
LIN {X 0,Y 652.65,Z 1136.578,A -85,B 0,C 180,E1 5700.905,E2 5700.905} C_VEL
LIN {X 0,Y 658.77,Z 1070.408,A -85,B 0,C 180,E1 5705.664,E2 5705.664} C_VEL
LIN {X 0,Y 664.46,Z 999.878,A -85,B 0,C 180,E1 5709.06,E2 5709.06} C_VEL
LIN {X 0,Y 668.481,Z 923.996,A -85,B 0,C 180,E1 5711.232,E2 5711.232} C_VEL
LIN {X 0,Y 667.985,Z 885.916,A -85,B 0,C 180,E1 5711.945,E2 5711.945} C_VEL
LIN {X 0,Y 642.393,Z 839.06,A -85,B 0,C 180,E1 5714.96,E2 5714.96} C_VEL
LIN {X 0,Y 642.461,Z 839.06,A -85,B 0,C 180,E1 5722.924,E2 5722.924} C_VEL
LIN {X 0,Y 642.644,Z 839.06,A -85,B 0,C 180,E1 5731.01,E2 5731.01} C_VEL
LIN {X 0,Y 642.078,Z 839.06,A -85,B 0,C 180,E1 5739.057,E2 5739.057} C_VEL
LIN {X 0,Y 642.486,Z 839.06,A -85,B 0,C 180,E1 5745.604,E2 5745.604} C_VEL
LIN {X 0,Y 642.887,Z 839.06,A -85,B 0,C 180,E1 5752.503,E2 5752.503} C_VEL
LIN {X 0,Y 642.874,Z 839.06,A -85,B 0,C 180,E1 5760.637,E2 5760.637} C_VEL
LIN {X 0,Y 642.535,Z 839.06,A -85,B 0,C 180,E1 5768.789,E2 5768.789} C_VEL
LIN {X 0,Y 642.299,Z 839.06,A -85,B 0,C 180,E1 5776.813,E2 5776.813} C_VEL
LIN {X 0,Y 642.397,Z 839.06,A -85,B 0,C 180,E1 5784.517,E2 5784.517} C_VEL
LIN {X 0,Y 642.175,Z 839.06,A -85,B 0,C 180,E1 5792.94,E2 5792.94} C_VEL
LIN {X 0,Y 642.14,Z 839.06,A -85,B 0,C 180,E1 5800.471,E2 5800.471} C_VEL
LIN {X 0,Y 642.492,Z 840.139,A -85,B 0,C 180,E1 5805.692,E2 5805.692} C_VEL
LIN {X 0,Y 668.761,Z 891.908,A -85,B 0,C 180,E1 5808.698,E2 5808.698} C_VEL
LIN {X 0,Y 664.974,Z 962.609,A -85,B 0,C 180,E1 5810.616,E2 5810.616} C_VEL
LIN {X 0,Y 659.322,Z 1034.286,A -85,B 0,C 180,E1 5813.929,E2 5813.929} C_VEL
LIN {X 0,Y 653.015,Z 1101.915,A -85,B 0,C 180,E1 5818.638,E2 5818.638} C_VEL
LIN {X 0,Y 647.977,Z 1158.621,A -85,B 0,C 180,E1 5824.314,E2 5824.314} C_VEL
LIN {X 0,Y 644.893,Z 1201.702,A -85,B 0,C 180,E1 5830.399,E2 5830.399} C_VEL
LIN {X 0,Y 643.358,Z 1231.98,A -85,B 0,C 180,E1 5836.698,E2 5836.698} C_VEL
LIN {X 0,Y 643.016,Z 1249.244,A -85,B 0,C 180,E1 5842.539,E2 5842.539} C_VEL
LIN {X 0,Y 642.95,Z 1256.412,A -85,B 0,C 180,E1 5847.97,E2 5847.97} C_VEL
LIN {X 0,Y 643.244,Z 1255.316,A -85,B 0,C 180,E1 5853.382,E2 5853.382} C_VEL
LIN {X 0,Y 643.249,Z 1244.037,A -85,B 0,C 180,E1 5859.509,E2 5859.509} C_VEL
LIN {X 0,Y 643.891,Z 1219.834,A -85,B 0,C 180,E1 5866.083,E2 5866.083} C_VEL
LIN {X 0,Y 646.25,Z 1181.835,A -85,B 0,C 180,E1 5872.582,E2 5872.582} C_VEL
LIN {X 0,Y 650.531,Z 1130.217,A -85,B 0,C 180,E1 5878.684,E2 5878.684} C_VEL
LIN {X 0,Y 656.299,Z 1067.911,A -85,B 0,C 180,E1 5883.859,E2 5883.859} C_VEL
LIN {X 0,Y 662.444,Z 997.551,A -85,B 0,C 180,E1 5887.862,E2 5887.862} C_VEL
LIN {X 0,Y 667.276,Z 923.601,A -85,B 0,C 180,E1 5890.511,E2 5890.511} C_VEL
LIN {X 0,Y 667.376,Z 885.659,A -85,B 0,C 180,E1 5891.454,E2 5891.454} C_VEL
LIN {X 0,Y 642.36,Z 839.06,A -85,B 0,C 180,E1 5894.247,E2 5894.247} C_VEL
LIN {X 0,Y 642.369,Z 839.06,A -85,B 0,C 180,E1 5903.016,E2 5903.016} C_VEL
LIN {X 0,Y 642.503,Z 839.06,A -85,B 0,C 180,E1 5911.092,E2 5911.092} C_VEL
LIN {X 0,Y 642.335,Z 839.06,A -85,B 0,C 180,E1 5920.013,E2 5920.013} C_VEL
LIN {X 0,Y 642.833,Z 839.06,A -85,B 0,C 180,E1 5928.539,E2 5928.539} C_VEL
LIN {X 0,Y 642.484,Z 839.06,A -85,B 0,C 180,E1 5936.654,E2 5936.654} C_VEL
LIN {X 0,Y 642.47,Z 839.06,A -85,B 0,C 180,E1 5942.069,E2 5942.069} C_VEL
LIN {X 0,Y 642.421,Z 839.06,A -85,B 0,C 180,E1 5948.87,E2 5948.87} C_VEL
LIN {X 0,Y 642.217,Z 839.06,A -85,B 0,C 180,E1 5957.216,E2 5957.216} C_VEL
LIN {X 0,Y 642.393,Z 839.06,A -85,B 0,C 180,E1 5964.518,E2 5964.518} C_VEL
LIN {X 0,Y 642.159,Z 839.06,A -85,B 0,C 180,E1 5972.94,E2 5972.94} C_VEL
LIN {X 0,Y 642.133,Z 839.06,A -85,B 0,C 180,E1 5980.107,E2 5980.107} C_VEL
LIN {X 0,Y 634.195,Z 839.06,A -85,B 0,C 180,E1 5983.194,E2 5983.194} C_VEL
LIN {X 0,Y 634.642,Z 841.072,A -85,B 0,C 180,E1 5984.591,E2 5984.591} C_VEL
LIN {X 0,Y 663.255,Z 893.952,A -85,B 0,C 180,E1 5987.804,E2 5987.804} C_VEL
LIN {X 0,Y 660.059,Z 972.1,A -85,B 0,C 180,E1 5989.519,E2 5989.519} C_VEL
LIN {X 0,Y 654.454,Z 1044.517,A -85,B 0,C 180,E1 5992.475,E2 5992.475} C_VEL
LIN {X 0,Y 647.795,Z 1113.632,A -85,B 0,C 180,E1 5996.834,E2 5996.834} C_VEL
LIN {X 0,Y 641.808,Z 1173.914,A -85,B 0,C 180,E1 6002.342,E2 6002.342} C_VEL
LIN {X 0,Y 637.641,Z 1221.562,A -85,B 0,C 180,E1 6008.528,E2 6008.528} C_VEL
LIN {X 0,Y 635.686,Z 1254.549,A -85,B 0,C 180,E1 6014.735,E2 6014.735} C_VEL
LIN {X 0,Y 635.033,Z 1276.004,A -85,B 0,C 180,E1 6021.061,E2 6021.061} C_VEL
LIN {X 0,Y 634.82,Z 1285.351,A -85,B 0,C 180,E1 6026.573,E2 6026.573} C_VEL
LIN {X 0,Y 634.744,Z 1286.378,A -85,B 0,C 180,E1 6032.056,E2 6032.056} C_VEL
LIN {X 0,Y 634.887,Z 1279.146,A -85,B 0,C 180,E1 6037.557,E2 6037.557} C_VEL
LIN {X 0,Y 635.375,Z 1261.806,A -85,B 0,C 180,E1 6043.472,E2 6043.472} C_VEL
LIN {X 0,Y 636.885,Z 1232.49,A -85,B 0,C 180,E1 6049.669,E2 6049.669} C_VEL
LIN {X 0,Y 640.316,Z 1190.286,A -85,B 0,C 180,E1 6055.758,E2 6055.758} C_VEL
LIN {X 0,Y 645.766,Z 1133.241,A -85,B 0,C 180,E1 6061.584,E2 6061.584} C_VEL
LIN {X 0,Y 652.56,Z 1065.451,A -85,B 0,C 180,E1 6066.387,E2 6066.387} C_VEL
LIN {X 0,Y 658.606,Z 994.291,A -85,B 0,C 180,E1 6069.72,E2 6069.72} C_VEL
LIN {X 0,Y 662.612,Z 920.721,A -85,B 0,C 180,E1 6071.751,E2 6071.751} C_VEL
LIN {X 0,Y 662.005,Z 889.293,A -85,B 0,C 180,E1 6072.363,E2 6072.363} C_VEL
LIN {X 0,Y 634.384,Z 839.06,A -85,B 0,C 180,E1 6075.623,E2 6075.623} C_VEL
LIN {X 0,Y 634.408,Z 839.06,A -85,B 0,C 180,E1 6084.084,E2 6084.084} C_VEL
LIN {X 0,Y 634.604,Z 839.06,A -85,B 0,C 180,E1 6092.168,E2 6092.168} C_VEL
LIN {X 0,Y 634.18,Z 839.06,A -85,B 0,C 180,E1 6101.009,E2 6101.009} C_VEL
LIN {X 0,Y 634.623,Z 839.06,A -85,B 0,C 180,E1 6109.631,E2 6109.631} C_VEL
LIN {X 0,Y 635.564,Z 839.06,A -85,B 0,C 180,E1 6119.277,E2 6119.277} C_VEL
LIN {X 0,Y 635.003,Z 839.06,A -85,B 0,C 180,E1 6127.511,E2 6127.511} C_VEL
LIN {X 0,Y 634.519,Z 839.06,A -85,B 0,C 180,E1 6135.92,E2 6135.92} C_VEL
LIN {X 0,Y 634.369,Z 839.06,A -85,B 0,C 180,E1 6144.699,E2 6144.699} C_VEL
LIN {X 0,Y 634.203,Z 839.06,A -85,B 0,C 180,E1 6152.519,E2 6152.519} C_VEL
LIN {X 0,Y 634.132,Z 839.06,A -85,B 0,C 180,E1 6161.091,E2 6161.091} C_VEL
LIN {X 0,Y 634.51,Z 840.197,A -85,B 0,C 180,E1 6164.982,E2 6164.982} C_VEL
LIN {X 0,Y 662.626,Z 894.704,A -85,B 0,C 180,E1 6168.294,E2 6168.294} C_VEL
LIN {X 0,Y 658.497,Z 965.042,A -85,B 0,C 180,E1 6170.26,E2 6170.26} C_VEL
LIN {X 0,Y 652.472,Z 1036.132,A -85,B 0,C 180,E1 6173.607,E2 6173.607} C_VEL
LIN {X 0,Y 645.729,Z 1103.28,A -85,B 0,C 180,E1 6178.372,E2 6178.372} C_VEL
LIN {X 0,Y 640.272,Z 1160.272,A -85,B 0,C 180,E1 6184.193,E2 6184.193} C_VEL
LIN {X 0,Y 637.015,Z 1202.67,A -85,B 0,C 180,E1 6190.323,E2 6190.323} C_VEL
LIN {X 0,Y 635.437,Z 1231.977,A -85,B 0,C 180,E1 6196.53,E2 6196.53} C_VEL
LIN {X 0,Y 635.045,Z 1249.243,A -85,B 0,C 180,E1 6202.444,E2 6202.444} C_VEL
LIN {X 0,Y 634.954,Z 1256.412,A -85,B 0,C 180,E1 6207.944,E2 6207.944} C_VEL
LIN {X 0,Y 635.22,Z 1255.317,A -85,B 0,C 180,E1 6213.425,E2 6213.425} C_VEL
LIN {X 0,Y 635.236,Z 1244.038,A -85,B 0,C 180,E1 6219.63,E2 6219.63} C_VEL
LIN {X 0,Y 635.945,Z 1219.837,A -85,B 0,C 180,E1 6226.289,E2 6226.289} C_VEL
LIN {X 0,Y 638.466,Z 1182.964,A -85,B 0,C 180,E1 6232.703,E2 6232.703} C_VEL
LIN {X 0,Y 642.938,Z 1132.815,A -85,B 0,C 180,E1 6238.773,E2 6238.773} C_VEL
LIN {X 0,Y 649.138,Z 1070.705,A -85,B 0,C 180,E1 6244.072,E2 6244.072} C_VEL
LIN {X 0,Y 655.687,Z 1001.227,A -85,B 0,C 180,E1 6248.13,E2 6248.13} C_VEL
LIN {X 0,Y 660.857,Z 927.558,A -85,B 0,C 180,E1 6250.86,E2 6250.86} C_VEL
LIN {X 0,Y 661.301,Z 889.122,A -85,B 0,C 180,E1 6251.843,E2 6251.843} C_VEL
LIN {X 0,Y 634.424,Z 839.06,A -85,B 0,C 180,E1 6255.07,E2 6255.07} C_VEL
LIN {X 0,Y 634.261,Z 839.06,A -85,B 0,C 180,E1 6264.171,E2 6264.171} C_VEL
LIN {X 0,Y 634.356,Z 839.06,A -85,B 0,C 180,E1 6272.245,E2 6272.245} C_VEL
LIN {X 0,Y 634.364,Z 839.06,A -85,B 0,C 180,E1 6279.751,E2 6279.751} C_VEL
LIN {X 0,Y 634.818,Z 839.06,A -85,B 0,C 180,E1 6288.319,E2 6288.319} C_VEL
LIN {X 0,Y 634.472,Z 839.06,A -85,B 0,C 180,E1 6296.612,E2 6296.612} C_VEL
LIN {X 0,Y 634.464,Z 839.06,A -85,B 0,C 180,E1 6302.095,E2 6302.095} C_VEL
LIN {X 0,Y 634.402,Z 839.06,A -85,B 0,C 180,E1 6308.983,E2 6308.983} C_VEL
LIN {X 0,Y 634.494,Z 839.06,A -85,B 0,C 180,E1 6316.002,E2 6316.002} C_VEL
LIN {X 0,Y 634.359,Z 839.06,A -85,B 0,C 180,E1 6324.786,E2 6324.786} C_VEL
LIN {X 0,Y 634.178,Z 839.06,A -85,B 0,C 180,E1 6332.614,E2 6332.614} C_VEL
LIN {X 0,Y 634.094,Z 839.06,A -85,B 0,C 180,E1 6341.199,E2 6341.199} C_VEL
LIN {X 0,Y 634.195,Z 839.06,A -85,B 0,C 180,E1 6343.194,E2 6343.194} C_VEL
LIN {X 0,Y 635.425,Z 847.898,A -85,B 0,C 180,E1 6344.499,E2 6344.499} C_VEL
LIN {X 0,Y 640.02,Z 863.387,A -85,B 0,C 180,E1 6345.418,E2 6345.418} C_VEL
LIN {X 0,Y 657.242,Z 897.294,A -85,B 0,C 180,E1 6347.384,E2 6347.384} C_VEL
LIN {X 0,Y 653.683,Z 975.038,A -85,B 0,C 180,E1 6349.154,E2 6349.154} C_VEL
LIN {X 0,Y 647.749,Z 1046.748,A -85,B 0,C 180,E1 6352.144,E2 6352.144} C_VEL
LIN {X 0,Y 640.655,Z 1115.256,A -85,B 0,C 180,E1 6356.547,E2 6356.547} C_VEL
LIN {X 0,Y 634.228,Z 1175.537,A -85,B 0,C 180,E1 6362.176,E2 6362.176} C_VEL
LIN {X 0,Y 629.782,Z 1222.899,A -85,B 0,C 180,E1 6368.47,E2 6368.47} C_VEL
LIN {X 0,Y 627.724,Z 1255.844,A -85,B 0,C 180,E1 6374.84,E2 6374.84} C_VEL
LIN {X 0,Y 627.026,Z 1276.005,A -85,B 0,C 180,E1 6380.946,E2 6380.946} C_VEL
LIN {X 0,Y 626.825,Z 1285.35,A -85,B 0,C 180,E1 6386.529,E2 6386.529} C_VEL
LIN {X 0,Y 626.748,Z 1286.378,A -85,B 0,C 180,E1 6392.083,E2 6392.083} C_VEL
LIN {X 0,Y 626.896,Z 1279.146,A -85,B 0,C 180,E1 6397.654,E2 6397.654} C_VEL
LIN {X 0,Y 627.417,Z 1261.805,A -85,B 0,C 180,E1 6403.646,E2 6403.646} C_VEL
LIN {X 0,Y 629.023,Z 1233.078,A -85,B 0,C 180,E1 6409.816,E2 6409.816} C_VEL
LIN {X 0,Y 632.708,Z 1191.09,A -85,B 0,C 180,E1 6415.988,E2 6415.988} C_VEL
LIN {X 0,Y 638.627,Z 1133.723,A -85,B 0,C 180,E1 6421.933,E2 6421.933} C_VEL
LIN {X 0,Y 645.741,Z 1066.963,A -85,B 0,C 180,E1 6426.732,E2 6426.732} C_VEL
LIN {X 0,Y 652.146,Z 997.328,A -85,B 0,C 180,E1 6430.057,E2 6430.057} C_VEL
LIN {X 0,Y 656.505,Z 923.898,A -85,B 0,C 180,E1 6432.156,E2 6432.156} C_VEL
LIN {X 0,Y 655.908,Z 892.197,A -85,B 0,C 180,E1 6432.808,E2 6432.808} C_VEL
LIN {X 0,Y 626.317,Z 839.06,A -85,B 0,C 180,E1 6436.284,E2 6436.284} C_VEL
LIN {X 0,Y 626.367,Z 839.06,A -85,B 0,C 180,E1 6445.256,E2 6445.256} C_VEL
LIN {X 0,Y 626.605,Z 839.06,A -85,B 0,C 180,E1 6453.344,E2 6453.344} C_VEL
LIN {X 0,Y 626.538,Z 839.06,A -85,B 0,C 180,E1 6463.157,E2 6463.157} C_VEL
LIN {X 0,Y 626.895,Z 839.06,A -85,B 0,C 180,E1 6472.311,E2 6472.311} C_VEL
LIN {X 0,Y 626.884,Z 839.06,A -85,B 0,C 180,E1 6480.654,E2 6480.654} C_VEL
LIN {X 0,Y 626.485,Z 839.06,A -85,B 0,C 180,E1 6489.016,E2 6489.016} C_VEL
LIN {X 0,Y 626.303,Z 839.06,A -85,B 0,C 180,E1 6496.772,E2 6496.772} C_VEL
LIN {X 0,Y 626.321,Z 839.06,A -85,B 0,C 180,E1 6505.038,E2 6505.038} C_VEL
LIN {X 0,Y 626.111,Z 839.06,A -85,B 0,C 180,E1 6513.225,E2 6513.225} C_VEL
LIN {X 0,Y 626.09,Z 839.06,A -85,B 0,C 180,E1 6521.736,E2 6521.736} C_VEL
LIN {X 0,Y 626.395,Z 840.294,A -85,B 0,C 180,E1 6524.231,E2 6524.231} C_VEL
LIN {X 0,Y 656.522,Z 897.917,A -85,B 0,C 180,E1 6527.891,E2 6527.891} C_VEL
LIN {X 0,Y 652.054,Z 967.5,A -85,B 0,C 180,E1 6529.899,E2 6529.899} C_VEL
LIN {X 0,Y 645.51,Z 1038.829,A -85,B 0,C 180,E1 6533.335,E2 6533.335} C_VEL
LIN {X 0,Y 638.358,Z 1105.695,A -85,B 0,C 180,E1 6538.195,E2 6538.195} C_VEL
